gfCNCPoint6[6065] = {X 274.4972, Y 101.6039, Z -8.0000, A 0.000, B 0.000, C 0.000 }
gfCNCPoint6[6066] = {X 273.7387, Y 101.1273, Z -8.0000, A 0.000, B 0.000, C 0.000 }
gfCNCPoint6[6067] = {X 273.1054, Y 100.4940, Z -8.0000, A 0.000, B 0.000, C 0.000 }
gfCNCPoint6[6068] = {X 272.6288, Y 99.7355, Z -8.0000, A 0.000, B 0.000, C 0.000 }
gfCNCPoint6[6069] = {X 272.3330, Y 98.8901, Z -8.0000, A 0.000, B 0.000, C 0.000 }
gfCNCPoint6[6070] = {X 272.2327, Y 98.0000, Z -8.0000, A 0.000, B 0.000, C 0.000 }
gfCNCPoint6[6071] = {X 272.2329, Y 97.0232, Z -8.0000, A 0.000, B 0.000, C 0.000 }
gfCNCPoint6[6072] = {X 272.3321, Y 96.1797, Z -8.0000, A 0.000, B 0.000, C 0.000 }
gfCNCPoint6[6073] = {X 272.6072, Y 95.3761, Z -8.0000, A 0.000, B 0.000, C 0.000 }
gfCNCPoint6[6074] = {X 273.0457, Y 94.6486, Z -8.0000, A 0.000, B 0.000, C 0.000 }
gfCNCPoint6[6075] = {X 273.6280, Y 94.0302, Z -8.0000, A 0.000, B 0.000, C 0.000 }
gfCNCPoint6[6076] = {X 274.3277, Y 93.5487, Z -8.0000, A 0.000, B 0.000, C 0.000 }
gfCNCPoint6[6077] = {X 275.1133, Y 93.2258, Z -8.0000, A 0.000, B 0.000, C 0.000 }
gfCNCPoint6[6078] = {X 275.9494, Y 93.0760, Z -8.0000, A 0.000, B 0.000, C 0.000 }
gfCNCPoint6[6079] = {X 275.9494, Y 85.3767, Z -8.0000, A 0.000, B 0.000, C 0.000 }
gfCNCPoint6[6080] = {X 262.6059, Y 80.1460, Z -8.0000, A 0.000, B 0.000, C 0.000 }
gfCNCPoint6[6081] = {X 237.4769, Y 96.4149, Z -8.0000, A 0.000, B 0.000, C 0.000 }
gfCNCPoint6[6082] = {X 237.4798, Y 97.0659, Z -8.0000, A 0.000, B 0.000, C 0.000 }
gfCNCPoint6[6083] = {X 237.4798, Y 98.0000, Z -8.0000, A 0.000, B 0.000, C 0.000 }
gfCNCPoint6[6084] = {X 237.3795, Y 98.8901, Z -8.0000, A 0.000, B 0.000, C 0.000 }
gfCNCPoint6[6085] = {X 237.0837, Y 99.7355, Z -8.0000, A 0.000, B 0.000, C 0.000 }
gfCNCPoint6[6086] = {X 236.6071, Y 100.4940, Z -8.0000, A 0.000, B 0.000, C 0.000 }
gfCNCPoint6[6087] = {X 235.9737, Y 101.1273, Z -8.0000, A 0.000, B 0.000, C 0.000 }
gfCNCPoint6[6088] = {X 235.2153, Y 101.6039, Z -8.0000, A 0.000, B 0.000, C 0.000 }
gfCNCPoint6[6089] = {X 234.3699, Y 101.8997, Z -8.0000, A 0.000, B 0.000, C 0.000 }
gfCNCPoint6[6090] = {X 233.4798, Y 102.0000, Z -8.0000, A 0.000, B 0.000, C 0.000 }
gfCNCPoint6[6091] = {X 214.1790, Y 102.0000, Z -8.0000, A 0.000, B 0.000, C 0.000 }
gfCNCPoint6[6092] = {X 213.7859, Y 101.9806, Z -8.0000, A 0.000, B 0.000, C 0.000 }
gfCNCPoint6[6093] = {X 213.3966, Y 101.9227, Z -8.0000, A 0.000, B 0.000, C 0.000 }
gfCNCPoint6[6094] = {X 213.0072, Y 101.9806, Z -8.0000, A 0.000, B 0.000, C 0.000 }
gfCNCPoint6[6095] = {X 212.6141, Y 102.0000, Z -8.0000, A 0.000, B 0.000, C 0.000 }
gfCNCPoint6[6096] = {X 194.9870, Y 102.0000, Z -8.0000, A 0.000, B 0.000, C 0.000 }
gfCNCPoint6[6097] = {X 194.0969, Y 101.8997, Z -8.0000, A 0.000, B 0.000, C 0.000 }
gfCNCPoint6[6098] = {X 193.2514, Y 101.6039, Z -8.0000, A 0.000, B 0.000, C 0.000 }
gfCNCPoint6[6099] = {X 192.4930, Y 101.1273, Z -8.0000, A 0.000, B 0.000, C 0.000 }
gfCNCPoint6[6100] = {X 191.8596, Y 100.4940, Z -8.0000, A 0.000, B 0.000, C 0.000 }
gfCNCPoint6[6101] = {X 191.3831, Y 99.7355, Z -8.0000, A 0.000, B 0.000, C 0.000 }
gfCNCPoint6[6102] = {X 191.0872, Y 98.8901, Z -8.0000, A 0.000, B 0.000, C 0.000 }
gfCNCPoint6[6103] = {X 190.9870, Y 98.0000, Z -8.0000, A 0.000, B 0.000, C 0.000 }
gfCNCPoint6[6104] = {X 190.9870, Y 97.0659, Z -8.0000, A 0.000, B 0.000, C 0.000 }
gfCNCPoint6[6105] = {X 191.0804, Y 96.2066, Z -8.0000, A 0.000, B 0.000, C 0.000 }
gfCNCPoint6[6106] = {X 191.3562, Y 95.3874, Z -8.0000, A 0.000, B 0.000, C 0.000 }
gfCNCPoint6[6107] = {X 191.8015, Y 94.6466, Z -8.0000, A 0.000, B 0.000, C 0.000 }
gfCNCPoint6[6108] = {X 191.9051, Y 94.5173, Z -8.0000, A 0.000, B 0.000, C 0.000 }
gfCNCPoint6[6109] = {X 192.0141, Y 94.3923, Z -8.0000, A 0.000, B 0.000, C 0.000 }
gfCNCPoint6[6110] = {X 188.7055, Y 90.7802, Z -8.0000, A 0.000, B 0.000, C 0.000 }
gfCNCPoint6[6111] = {X 149.9476, Y 90.7802, Z -8.0000, A 0.000, B 0.000, C 0.000 }
gfCNCPoint6[6112] = {X 146.7195, Y 94.3565, Z -8.0000, A 0.000, B 0.000, C 0.000 }
gfCNCPoint6[6113] = {X 147.1699, Y 94.9478, Z -8.0000, A 0.000, B 0.000, C 0.000 }
gfCNCPoint6[6114] = {X 147.5035, Y 95.6119, Z -8.0000, A 0.000, B 0.000, C 0.000 }
gfCNCPoint6[6115] = {X 147.7089, Y 96.3261, Z -8.0000, A 0.000, B 0.000, C 0.000 }
gfCNCPoint6[6116] = {X 147.7791, Y 97.0660, Z -8.0000, A 0.000, B 0.000, C 0.000 }
gfCNCPoint6[6117] = {X 147.7791, Y 98.0000, Z -8.0000, A 0.000, B 0.000, C 0.000 }
gfCNCPoint6[6118] = {X 147.6788, Y 98.8901, Z -8.0000, A 0.000, B 0.000, C 0.000 }
gfCNCPoint6[6119] = {X 147.3830, Y 99.7355, Z -8.0000, A 0.000, B 0.000, C 0.000 }
gfCNCPoint6[6120] = {X 146.9064, Y 100.4940, Z -8.0000, A 0.000, B 0.000, C 0.000 }
gfCNCPoint6[6121] = {X 146.2731, Y 101.1273, Z -8.0000, A 0.000, B 0.000, C 0.000 }
gfCNCPoint6[6122] = {X 145.5146, Y 101.6039, Z -8.0000, A 0.000, B 0.000, C 0.000 }
gfCNCPoint6[6123] = {X 144.6692, Y 101.8997, Z -8.0000, A 0.000, B 0.000, C 0.000 }
gfCNCPoint6[6124] = {X 143.7791, Y 102.0000, Z -8.0000, A 0.000, B 0.000, C 0.000 }
gfCNCPoint6[6125] = {X 125.0000, Y 102.0000, Z -8.0000, A 0.000, B 0.000, C 0.000 }
gfCNCPoint6[6126] = {X 124.1099, Y 101.8997, Z -8.0000, A 0.000, B 0.000, C 0.000 }
gfCNCPoint6[6127] = {X 123.2645, Y 101.6039, Z -8.0000, A 0.000, B 0.000, C 0.000 }
gfCNCPoint6[6128] = {X 122.5060, Y 101.1273, Z -8.0000, A 0.000, B 0.000, C 0.000 }
gfCNCPoint6[6129] = {X 121.8727, Y 100.4940, Z -8.0000, A 0.000, B 0.000, C 0.000 }
gfCNCPoint6[6130] = {X 121.3961, Y 99.7355, Z -8.0000, A 0.000, B 0.000, C 0.000 }
gfCNCPoint6[6131] = {X 121.1003, Y 98.8901, Z -8.0000, A 0.000, B 0.000, C 0.000 }
gfCNCPoint6[6132] = {X 121.0000, Y 98.0000, Z -8.0000, A 0.000, B 0.000, C 0.000 }
gfCNCPoint6[6133] = {X 121.0000, Y 97.0659, Z -8.0000, A 0.000, B 0.000, C 0.000 }
gfCNCPoint6[6134] = {X 121.0981, Y 96.1853, Z -8.0000, A 0.000, B 0.000, C 0.000 }
gfCNCPoint6[6135] = {X 121.3877, Y 95.3479, Z -8.0000, A 0.000, B 0.000, C 0.000 }
gfCNCPoint6[6136] = {X 121.8546, Y 94.5948, Z -8.0000, A 0.000, B 0.000, C 0.000 }
gfCNCPoint6[6137] = {X 122.4758, Y 93.9629, Z -8.0000, A 0.000, B 0.000, C 0.000 }
gfCNCPoint6[6138] = {X 123.2209, Y 93.4834, Z -8.0000, A 0.000, B 0.000, C 0.000 }
gfCNCPoint6[6139] = {X 124.0533, Y 93.1796, Z -8.0000, A 0.000, B 0.000, C 0.000 }
gfCNCPoint6[6140] = {X 124.9321, Y 93.0665, Z -8.0000, A 0.000, B 0.000, C 0.000 }
gfCNCPoint6[6141] = {X 124.9746, Y 93.0367, Z -8.0000, A 0.000, B 0.000, C 0.000 }
gfCNCPoint6[6142] = {X 125.4940, Y 92.9596, Z -8.0000, A 0.000, B 0.000, C 0.000 }
gfCNCPoint6[6143] = {X 126.3820, Y 92.8084, Z -8.0000, A 0.000, B 0.000, C 0.000 }
gfCNCPoint6[6144] = {X 127.2570, Y 92.5949, Z -8.0000, A 0.000, B 0.000, C 0.000 }
gfCNCPoint6[6145] = {X 128.4861, Y 91.4437, Z -8.0000, A 0.000, B 0.000, C 0.000 }
gfCNCPoint6[6146] = {X 129.6489, Y 90.2255, Z -8.0000, A 0.000, B 0.000, C 0.000 }
gfCNCPoint6[6147] = {X 140.9159, Y 77.8537, Z -8.0000, A 0.000, B 0.000, C 0.000 }
gfCNCPoint6[6148] = {X 137.8994, Y 75.1065, Z -8.0000, A 0.000, B 0.000, C 0.000 }
gfCNCPoint6[6149] = {X 137.8994, Y 75.1065, Z -5.0000, A 0.000, B 0.000, C 0.000 }
gfCNCPoint6[6150] = {X 137.8994, Y 75.1065, Z 11.0000, A 0.000, B 0.000, C 0.000 }
gfCNCPoint6[6151] = {X 165.2857, Y 38.5771, Z 11.0000, A 0.000, B 0.000, C 0.000 }
gfCNCPoint6[6152] = {X 165.2857, Y 38.5771, Z -5.0000, A 0.000, B 0.000, C 0.000 }
gfCNCPoint6[6153] = {X 165.2857, Y 38.5771, Z -8.0000, A 0.000, B 0.000, C 0.000 }
gfCNCPoint6[6154] = {X 169.3150, Y 37.9356, Z -8.0000, A 0.000, B 0.000, C 0.000 }
gfCNCPoint6[6155] = {X 169.2595, Y 37.5870, Z -8.0000, A 0.000, B 0.000, C 0.000 }
gfCNCPoint6[6156] = {X 169.1010, Y 35.9822, Z -8.0000, A 0.000, B 0.000, C 0.000 }
gfCNCPoint6[6157] = {X 169.1179, Y 34.3697, Z -8.0000, A 0.000, B 0.000, C 0.000 }
gfCNCPoint6[6158] = {X 169.3102, Y 32.7686, Z -8.0000, A 0.000, B 0.000, C 0.000 }
gfCNCPoint6[6159] = {X 169.6755, Y 31.1979, Z -8.0000, A 0.000, B 0.000, C 0.000 }
gfCNCPoint6[6160] = {X 170.2095, Y 29.6763, Z -8.0000, A 0.000, B 0.000, C 0.000 }
gfCNCPoint6[6161] = {X 170.8480, Y 28.3694, Z -8.0000, A 0.000, B 0.000, C 0.000 }
gfCNCPoint6[6162] = {X 171.6556, Y 27.1596, Z -8.0000, A 0.000, B 0.000, C 0.000 }
gfCNCPoint6[6163] = {X 172.6177, Y 26.0688, Z -8.0000, A 0.000, B 0.000, C 0.000 }
gfCNCPoint6[6164] = {X 173.7171, Y 25.1164, Z -8.0000, A 0.000, B 0.000, C 0.000 }
gfCNCPoint6[6165] = {X 174.9340, Y 24.3195, Z -8.0000, A 0.000, B 0.000, C 0.000 }
gfCNCPoint6[6166] = {X 174.1517, Y 23.9319, Z -8.0000, A 0.000, B 0.000, C 0.000 }
gfCNCPoint6[6167] = {X 173.4633, Y 23.3948, Z -8.0000, A 0.000, B 0.000, C 0.000 }
gfCNCPoint6[6168] = {X 172.8970, Y 22.7303, Z -8.0000, A 0.000, B 0.000, C 0.000 }
gfCNCPoint6[6169] = {X 172.4758, Y 21.9655, Z -8.0000, A 0.000, B 0.000, C 0.000 }
gfCNCPoint6[6170] = {X 169.8405, Y 15.5121, Z -8.0000, A 0.000, B 0.000, C 0.000 }
gfCNCPoint6[6171] = {X 169.5912, Y 14.6607, Z -8.0000, A 0.000, B 0.000, C 0.000 }
gfCNCPoint6[6172] = {X 169.5212, Y 13.7764, Z -8.0000, A 0.000, B 0.000, C 0.000 }
gfCNCPoint6[6173] = {X 169.6332, Y 12.8964, Z -8.0000, A 0.000, B 0.000, C 0.000 }
gfCNCPoint6[6174] = {X 169.9226, Y 12.0578, Z -8.0000, A 0.000, B 0.000, C 0.000 }
gfCNCPoint6[6175] = {X 170.3773, Y 11.2960, Z -8.0000, A 0.000, B 0.000, C 0.000 }
gfCNCPoint6[6176] = {X 170.9779, Y 10.6432, Z -8.0000, A 0.000, B 0.000, C 0.000 }
gfCNCPoint6[6177] = {X 171.6992, Y 10.1268, Z -8.0000, A 0.000, B 0.000, C 0.000 }
gfCNCPoint6[6178] = {X 172.3295, Y 9.7674, Z -8.0000, A 0.000, B 0.000, C 0.000 }
gfCNCPoint6[6179] = {X 173.1918, Y 9.4018, Z -8.0000, A 0.000, B 0.000, C 0.000 }
gfCNCPoint6[6180] = {X 174.1126, Y 9.2307, Z -8.0000, A 0.000, B 0.000, C 0.000 }
gfCNCPoint6[6181] = {X 175.0486, Y 9.2620, Z -8.0000, A 0.000, B 0.000, C 0.000 }
gfCNCPoint6[6182] = {X 175.9559, Y 9.4943, Z -8.0000, A 0.000, B 0.000, C 0.000 }
gfCNCPoint6[6183] = {X 177.1286, Y 9.0434, Z -8.0000, A 0.000, B 0.000, C 0.000 }
gfCNCPoint6[6184] = {X 179.2966, Y 8.2457, Z -8.0000, A 0.000, B 0.000, C 0.000 }
gfCNCPoint6[6185] = {X 181.5326, Y 7.6654, Z -8.0000, A 0.000, B 0.000, C 0.000 }
gfCNCPoint6[6186] = {X 183.8149, Y 7.3083, Z -8.0000, A 0.000, B 0.000, C 0.000 }
gfCNCPoint6[6187] = {X 186.1213, Y 7.1778, Z -8.0000, A 0.000, B 0.000, C 0.000 }
gfCNCPoint6[6188] = {X 188.4294, Y 7.2751, Z -8.0000, A 0.000, B 0.000, C 0.000 }
gfCNCPoint6[6189] = {X 190.7166, Y 7.5994, Z -8.0000, A 0.000, B 0.000, C 0.000 }
gfCNCPoint6[6190] = {X 192.3080, Y 7.9856, Z -8.0000, A 0.000, B 0.000, C 0.000 }
gfCNCPoint6[6191] = {X 193.8552, Y 8.5222, Z -8.0000, A 0.000, B 0.000, C 0.000 }
gfCNCPoint6[6192] = {X 195.3440, Y 9.2045, Z -8.0000, A 0.000, B 0.000, C 0.000 }
gfCNCPoint6[6193] = {X 196.7606, Y 10.0260, Z -8.0000, A 0.000, B 0.000, C 0.000 }
gfCNCPoint6[6194] = {X 198.0922, Y 10.9792, Z -8.0000, A 0.000, B 0.000, C 0.000 }
gfCNCPoint6[6195] = {X 199.1520, Y 11.9221, Z -8.0000, A 0.000, B 0.000, C 0.000 }
gfCNCPoint6[6196] = {X 200.1030, Y 12.9747, Z -8.0000, A 0.000, B 0.000, C 0.000 }
gfCNCPoint6[6197] = {X 200.9339, Y 14.1244, Z -8.0000, A 0.000, B 0.000, C 0.000 }
gfCNCPoint6[6198] = {X 201.6348, Y 15.3577, Z -8.0000, A 0.000, B 0.000, C 0.000 }
gfCNCPoint6[6199] = {X 202.1974, Y 16.6600, Z -8.0000, A 0.000, B 0.000, C 0.000 }
gfCNCPoint6[6200] = {X 202.6716, Y 18.3163, Z -8.0000, A 0.000, B 0.000, C 0.000 }
gfCNCPoint6[6201] = {X 202.9530, Y 20.0160, Z -8.0000, A 0.000, B 0.000, C 0.000 }
gfCNCPoint6[6202] = {X 203.0380, Y 21.7368, Z -8.0000, A 0.000, B 0.000, C 0.000 }
gfCNCPoint6[6203] = {X 202.9255, Y 23.4560, Z -8.0000, A 0.000, B 0.000, C 0.000 }
gfCNCPoint6[6204] = {X 202.6168, Y 25.1510, Z -8.0000, A 0.000, B 0.000, C 0.000 }
gfCNCPoint6[6205] = {X 202.1749, Y 26.5972, Z -8.0000, A 0.000, B 0.000, C 0.000 }
gfCNCPoint6[6206] = {X 201.5500, Y 27.9742, Z -8.0000, A 0.000, B 0.000, C 0.000 }
gfCNCPoint6[6207] = {X 200.7528, Y 29.2592, Z -8.0000, A 0.000, B 0.000, C 0.000 }
gfCNCPoint6[6208] = {X 199.7964, Y 30.4306, Z -8.0000, A 0.000, B 0.000, C 0.000 }
gfCNCPoint6[6209] = {X 198.6969, Y 31.4688, Z -8.0000, A 0.000, B 0.000, C 0.000 }
gfCNCPoint6[6210] = {X 199.4979, Y 31.8101, Z -8.0000, A 0.000, B 0.000, C 0.000 }
gfCNCPoint6[6211] = {X 200.2141, Y 32.3050, Z -8.0000, A 0.000, B 0.000, C 0.000 }
gfCNCPoint6[6212] = {X 200.8166, Y 32.9336, Z -8.0000, A 0.000, B 0.000, C 0.000 }
gfCNCPoint6[6213] = {X 201.2808, Y 33.6702, Z -8.0000, A 0.000, B 0.000, C 0.000 }
gfCNCPoint6[6214] = {X 204.3222, Y 39.9530, Z -8.0000, A 0.000, B 0.000, C 0.000 }
gfCNCPoint6[6215] = {X 204.6427, Y 40.8622, Z -8.0000, A 0.000, B 0.000, C 0.000 }
gfCNCPoint6[6216] = {X 204.7537, Y 41.8197, Z -8.0000, A 0.000, B 0.000, C 0.000 }
gfCNCPoint6[6217] = {X 204.6496, Y 42.7781, Z -8.0000, A 0.000, B 0.000, C 0.000 }
gfCNCPoint6[6218] = {X 204.3355, Y 43.6895, Z -8.0000, A 0.000, B 0.000, C 0.000 }
gfCNCPoint6[6219] = {X 203.8272, Y 44.5085, Z -8.0000, A 0.000, B 0.000, C 0.000 }
gfCNCPoint6[6220] = {X 203.1499, Y 45.1945, Z -8.0000, A 0.000, B 0.000, C 0.000 }
gfCNCPoint6[6221] = {X 202.6139, Y 45.6278, Z -8.0000, A 0.000, B 0.000, C 0.000 }
gfCNCPoint6[6222] = {X 201.9096, Y 46.0923, Z -8.0000, A 0.000, B 0.000, C 0.000 }
gfCNCPoint6[6223] = {X 201.1286, Y 46.4113, Z -8.0000, A 0.000, B 0.000, C 0.000 }
gfCNCPoint6[6224] = {X 200.3005, Y 46.5727, Z -8.0000, A 0.000, B 0.000, C 0.000 }
gfCNCPoint6[6225] = {X 199.4569, Y 46.5704, Z -8.0000, A 0.000, B 0.000, C 0.000 }
gfCNCPoint6[6226] = {X 198.6297, Y 46.4045, Z -8.0000, A 0.000, B 0.000, C 0.000 }
gfCNCPoint6[6227] = {X 196.5191, Y 47.5053, Z -8.0000, A 0.000, B 0.000, C 0.000 }
gfCNCPoint6[6228] = {X 194.3239, Y 48.4257, Z -8.0000, A 0.000, B 0.000, C 0.000 }
gfCNCPoint6[6229] = {X 192.0594, Y 49.1592, Z -8.0000, A 0.000, B 0.000, C 0.000 }
gfCNCPoint6[6230] = {X 189.8462, Y 49.6717, Z -8.0000, A 0.000, B 0.000, C 0.000 }
gfCNCPoint6[6231] = {X 187.5926, Y 49.9576, Z -8.0000, A 0.000, B 0.000, C 0.000 }
gfCNCPoint6[6232] = {X 185.3216, Y 50.0138, Z -8.0000, A 0.000, B 0.000, C 0.000 }
gfCNCPoint6[6233] = {X 183.0565, Y 49.8399, Z -8.0000, A 0.000, B 0.000, C 0.000 }
gfCNCPoint6[6234] = {X 180.8207, Y 49.4375, Z -8.0000, A 0.000, B 0.000, C 0.000 }
gfCNCPoint6[6235] = {X 178.9807, Y 48.9033, Z -8.0000, A 0.000, B 0.000, C 0.000 }
gfCNCPoint6[6236] = {X 177.2144, Y 48.1610, Z -8.0000, A 0.000, B 0.000, C 0.000 }
gfCNCPoint6[6237] = {X 175.5452, Y 47.2205, Z -8.0000, A 0.000, B 0.000, C 0.000 }
gfCNCPoint6[6238] = {X 173.9952, Y 46.0942, Z -8.0000, A 0.000, B 0.000, C 0.000 }
gfCNCPoint6[6239] = {X 172.8545, Y 45.0533, Z -8.0000, A 0.000, B 0.000, C 0.000 }
gfCNCPoint6[6240] = {X 171.8449, Y 43.8848, Z -8.0000, A 0.000, B 0.000, C 0.000 }
gfCNCPoint6[6241] = {X 170.9807, Y 42.6050, Z -8.0000, A 0.000, B 0.000, C 0.000 }
gfCNCPoint6[6242] = {X 170.2740, Y 41.2319, Z -8.0000, A 0.000, B 0.000, C 0.000 }
gfCNCPoint6[6243] = {X 169.7348, Y 39.7849, Z -8.0000, A 0.000, B 0.000, C 0.000 }
gfCNCPoint6[6244] = {X 169.3705, Y 38.2842, Z -8.0000, A 0.000, B 0.000, C 0.000 }
gfCNCPoint6[6245] = {X 169.3150, Y 37.9356, Z -8.0000, A 0.000, B 0.000, C 0.000 }
gfCNCPoint6[6246] = {X 165.3647, Y 38.5646, Z -8.0000, A 0.000, B 0.000, C 0.000 }
gfCNCPoint6[6247] = {X 169.3940, Y 37.9231, Z -8.0000, A 0.000, B 0.000, C 0.000 }
gfCNCPoint6[6248] = {X 169.3385, Y 37.5748, Z -8.0000, A 0.000, B 0.000, C 0.000 }
gfCNCPoint6[6249] = {X 169.1809, Y 35.9787, Z -8.0000, A 0.000, B 0.000, C 0.000 }
gfCNCPoint6[6250] = {X 169.1978, Y 34.3748, Z -8.0000, A 0.000, B 0.000, C 0.000 }
gfCNCPoint6[6251] = {X 169.3890, Y 32.7823, Z -8.0000, A 0.000, B 0.000, C 0.000 }
gfCNCPoint6[6252] = {X 169.7524, Y 31.2201, Z -8.0000, A 0.000, B 0.000, C 0.000 }
gfCNCPoint6[6253] = {X 170.2835, Y 29.7067, Z -8.0000, A 0.000, B 0.000, C 0.000 }
gfCNCPoint6[6254] = {X 170.9351, Y 28.3785, Z -8.0000, A 0.000, B 0.000, C 0.000 }
gfCNCPoint6[6255] = {X 171.7625, Y 27.1522, Z -8.0000, A 0.000, B 0.000, C 0.000 }
gfCNCPoint6[6256] = {X 172.7502, Y 26.0509, Z -8.0000, A 0.000, B 0.000, C 0.000 }
gfCNCPoint6[6257] = {X 173.8794, Y 25.0952, Z -8.0000, A 0.000, B 0.000, C 0.000 }
gfCNCPoint6[6258] = {X 175.1290, Y 24.3033, Z -8.0000, A 0.000, B 0.000, C 0.000 }
gfCNCPoint6[6259] = {X 174.3078, Y 23.9331, Z -8.0000, A 0.000, B 0.000, C 0.000 }
gfCNCPoint6[6260] = {X 173.5833, Y 23.3977, Z -8.0000, A 0.000, B 0.000, C 0.000 }
gfCNCPoint6[6261] = {X 172.9883, Y 22.7214, Z -8.0000, A 0.000, B 0.000, C 0.000 }
gfCNCPoint6[6262] = {X 172.5496, Y 21.9347, Z -8.0000, A 0.000, B 0.000, C 0.000 }
gfCNCPoint6[6263] = {X 169.9145, Y 15.4818, Z -8.0000, A 0.000, B 0.000, C 0.000 }
gfCNCPoint6[6264] = {X 169.6699, Y 14.6462, Z -8.0000, A 0.000, B 0.000, C 0.000 }
gfCNCPoint6[6265] = {X 169.6011, Y 13.7783, Z -8.0000, A 0.000, B 0.000, C 0.000 }
gfCNCPoint6[6266] = {X 169.7111, Y 12.9146, Z -8.0000, A 0.000, B 0.000, C 0.000 }
gfCNCPoint6[6267] = {X 169.9952, Y 12.0915, Z -8.0000, A 0.000, B 0.000, C 0.000 }
gfCNCPoint6[6268] = {X 170.4414, Y 11.3439, Z -8.0000, A 0.000, B 0.000, C 0.000 }
gfCNCPoint6[6269] = {X 171.0309, Y 10.7031, Z -8.0000, A 0.000, B 0.000, C 0.000 }
gfCNCPoint6[6270] = {X 171.7389, Y 10.1963, Z -8.0000, A 0.000, B 0.000, C 0.000 }
gfCNCPoint6[6271] = {X 172.3689, Y 9.8371, Z -8.0000, A 0.000, B 0.000, C 0.000 }
gfCNCPoint6[6272] = {X 173.2224, Y 9.4762, Z -8.0000, A 0.000, B 0.000, C 0.000 }
gfCNCPoint6[6273] = {X 174.1339, Y 9.3093, Z -8.0000, A 0.000, B 0.000, C 0.000 }
gfCNCPoint6[6274] = {X 175.0599, Y 9.3445, Z -8.0000, A 0.000, B 0.000, C 0.000 }
gfCNCPoint6[6275] = {X 175.9561, Y 9.5799, Z -8.0000, A 0.000, B 0.000, C 0.000 }
gfCNCPoint6[6276] = {X 177.1586, Y 9.1176, Z -8.0000, A 0.000, B 0.000, C 0.000 }
gfCNCPoint6[6277] = {X 179.3194, Y 8.3224, Z -8.0000, A 0.000, B 0.000, C 0.000 }
gfCNCPoint6[6278] = {X 181.5480, Y 7.7439, Z -8.0000, A 0.000, B 0.000, C 0.000 }
gfCNCPoint6[6279] = {X 183.8227, Y 7.3879, Z -8.0000, A 0.000, B 0.000, C 0.000 }
gfCNCPoint6[6280] = {X 186.1214, Y 7.2578, Z -8.0000, A 0.000, B 0.000, C 0.000 }
gfCNCPoint6[6281] = {X 188.4218, Y 7.3548, Z -8.0000, A 0.000, B 0.000, C 0.000 }
gfCNCPoint6[6282] = {X 190.7015, Y 7.6779, Z -8.0000, A 0.000, B 0.000, C 0.000 }
gfCNCPoint6[6283] = {X 192.2855, Y 8.0623, Z -8.0000, A 0.000, B 0.000, C 0.000 }
gfCNCPoint6[6284] = {X 193.8254, Y 8.5965, Z -8.0000, A 0.000, B 0.000, C 0.000 }
gfCNCPoint6[6285] = {X 195.3072, Y 9.2755, Z -8.0000, A 0.000, B 0.000, C 0.000 }
gfCNCPoint6[6286] = {X 196.7172, Y 10.0932, Z -8.0000, A 0.000, B 0.000, C 0.000 }
gfCNCPoint6[6287] = {X 198.0426, Y 11.0420, Z -8.0000, A 0.000, B 0.000, C 0.000 }
gfCNCPoint6[6288] = {X 199.0958, Y 11.9791, Z -8.0000, A 0.000, B 0.000, C 0.000 }
gfCNCPoint6[6289] = {X 200.0409, Y 13.0251, Z -8.0000, A 0.000, B 0.000, C 0.000 }
gfCNCPoint6[6290] = {X 200.8666, Y 14.1678, Z -8.0000, A 0.000, B 0.000, C 0.000 }
gfCNCPoint6[6291] = {X 201.5632, Y 15.3935, Z -8.0000, A 0.000, B 0.000, C 0.000 }
gfCNCPoint6[6292] = {X 202.1223, Y 16.6876, Z -8.0000, A 0.000, B 0.000, C 0.000 }
gfCNCPoint6[6293] = {X 202.5938, Y 18.3350, Z -8.0000, A 0.000, B 0.000, C 0.000 }
gfCNCPoint6[6294] = {X 202.8736, Y 20.0255, Z -8.0000, A 0.000, B 0.000, C 0.000 }
gfCNCPoint6[6295] = {X 202.9580, Y 21.7368, Z -8.0000, A 0.000, B 0.000, C 0.000 }
gfCNCPoint6[6296] = {X 202.8460, Y 23.4467, Z -8.0000, A 0.000, B 0.000, C 0.000 }
gfCNCPoint6[6297] = {X 202.5390, Y 25.1324, Z -8.0000, A 0.000, B 0.000, C 0.000 }
gfCNCPoint6[6298] = {X 202.0893, Y 26.5970, Z -8.0000, A 0.000, B 0.000, C 0.000 }
gfCNCPoint6[6299] = {X 201.4509, Y 27.9898, Z -8.0000, A 0.000, B 0.000, C 0.000 }
gfCNCPoint6[6300] = {X 200.6347, Y 29.2864, Z -8.0000, A 0.000, B 0.000, C 0.000 }
gfCNCPoint6[6301] = {X 199.6550, Y 30.4643, Z -8.0000, A 0.000, B 0.000, C 0.000 }
gfCNCPoint6[6302] = {X 198.5287, Y 31.5030, Z -8.0000, A 0.000, B 0.000, C 0.000 }
gfCNCPoint6[6303] = {X 199.3597, Y 31.8270, Z -8.0000, A 0.000, B 0.000, C 0.000 }
gfCNCPoint6[6304] = {X 200.1046, Y 32.3177, Z -8.0000, A 0.000, B 0.000, C 0.000 }
gfCNCPoint6[6305] = {X 200.7303, Y 32.9533, Z -8.0000, A 0.000, B 0.000, C 0.000 }
gfCNCPoint6[6306] = {X 201.2091, Y 33.7058, Z -8.0000, A 0.000, B 0.000, C 0.000 }
gfCNCPoint6[6307] = {X 204.2502, Y 39.9879, Z -8.0000, A 0.000, B 0.000, C 0.000 }
gfCNCPoint6[6308] = {X 204.5648, Y 40.8802, Z -8.0000, A 0.000, B 0.000, C 0.000 }
gfCNCPoint6[6309] = {X 204.6737, Y 41.8200, Z -8.0000, A 0.000, B 0.000, C 0.000 }
gfCNCPoint6[6310] = {X 204.5715, Y 42.7606, Z -8.0000, A 0.000, B 0.000, C 0.000 }
gfCNCPoint6[6311] = {X 204.2633, Y 43.6551, Z -8.0000, A 0.000, B 0.000, C 0.000 }
gfCNCPoint6[6312] = {X 203.7643, Y 44.4590, Z -8.0000, A 0.000, B 0.000, C 0.000 }
gfCNCPoint6[6313] = {X 203.0996, Y 45.1323, Z -8.0000, A 0.000, B 0.000, C 0.000 }
gfCNCPoint6[6314] = {X 202.5635, Y 45.5657, Z -8.0000, A 0.000, B 0.000, C 0.000 }
gfCNCPoint6[6315] = {X 201.8662, Y 46.0248, Z -8.0000, A 0.000, B 0.000, C 0.000 }
gfCNCPoint6[6316] = {X 201.0924, Y 46.3386, Z -8.0000, A 0.000, B 0.000, C 0.000 }
gfCNCPoint6[6317] = {X 200.2723, Y 46.4950, Z -8.0000, A 0.000, B 0.000, C 0.000 }
gfCNCPoint6[6318] = {X 199.4374, Y 46.4880, Z -8.0000, A 0.000, B 0.000, C 0.000 }
gfCNCPoint6[6319] = {X 198.6200, Y 46.3178, Z -8.0000, A 0.000, B 0.000, C 0.000 }
gfCNCPoint6[6320] = {X 196.5061, Y 47.4230, Z -8.0000, A 0.000, B 0.000, C 0.000 }
gfCNCPoint6[6321] = {X 194.3068, Y 48.3467, Z -8.0000, A 0.000, B 0.000, C 0.000 }
gfCNCPoint6[6322] = {X 192.0377, Y 49.0822, Z -8.0000, A 0.000, B 0.000, C 0.000 }
gfCNCPoint6[6323] = {X 189.8323, Y 49.5930, Z -8.0000, A 0.000, B 0.000, C 0.000 }
gfCNCPoint6[6324] = {X 187.5867, Y 49.8778, Z -8.0000, A 0.000, B 0.000, C 0.000 }
gfCNCPoint6[6325] = {X 185.3237, Y 49.9339, Z -8.0000, A 0.000, B 0.000, C 0.000 }
gfCNCPoint6[6326] = {X 183.0666, Y 49.7605, Z -8.0000, A 0.000, B 0.000, C 0.000 }
gfCNCPoint6[6327] = {X 180.8387, Y 49.3596, Z -8.0000, A 0.000, B 0.000, C 0.000 }
gfCNCPoint6[6328] = {X 179.0075, Y 48.8279, Z -8.0000, A 0.000, B 0.000, C 0.000 }
gfCNCPoint6[6329] = {X 177.2496, Y 48.0891, Z -8.0000, A 0.000, B 0.000, C 0.000 }
gfCNCPoint6[6330] = {X 175.5883, Y 47.1531, Z -8.0000, A 0.000, B 0.000, C 0.000 }
gfCNCPoint6[6331] = {X 174.0457, Y 46.0322, Z -8.0000, A 0.000, B 0.000, C 0.000 }
gfCNCPoint6[6332] = {X 172.9120, Y 44.9978, Z -8.0000, A 0.000, B 0.000, C 0.000 }
gfCNCPoint6[6333] = {X 171.9087, Y 43.8365, Z -8.0000, A 0.000, B 0.000, C 0.000 }
gfCNCPoint6[6334] = {X 171.0498, Y 42.5647, Z -8.0000, A 0.000, B 0.000, C 0.000 }
gfCNCPoint6[6335] = {X 170.3475, Y 41.2002, Z -8.0000, A 0.000, B 0.000, C 0.000 }
gfCNCPoint6[6336] = {X 169.8115, Y 39.7622, Z -8.0000, A 0.000, B 0.000, C 0.000 }
gfCNCPoint6[6337] = {X 169.4494, Y 38.2708, Z -8.0000, A 0.000, B 0.000, C 0.000 }
gfCNCPoint6[6338] = {X 169.3940, Y 37.9231, Z -8.0000, A 0.000, B 0.000, C 0.000 }
gfCNCPoint6[6339] = {X 165.4437, Y 38.5520, Z -8.0000, A 0.000, B 0.000, C 0.000 }
gfCNCPoint6[6340] = {X 169.4730, Y 37.9105, Z -8.0000, A 0.000, B 0.000, C 0.000 }
gfCNCPoint6[6341] = {X 169.4176, Y 37.5627, Z -8.0000, A 0.000, B 0.000, C 0.000 }
gfCNCPoint6[6342] = {X 169.2608, Y 35.9751, Z -8.0000, A 0.000, B 0.000, C 0.000 }
gfCNCPoint6[6343] = {X 169.2776, Y 34.3799, Z -8.0000, A 0.000, B 0.000, C 0.000 }
gfCNCPoint6[6344] = {X 169.4679, Y 32.7961, Z -8.0000, A 0.000, B 0.000, C 0.000 }
gfCNCPoint6[6345] = {X 169.8292, Y 31.2423, Z -8.0000, A 0.000, B 0.000, C 0.000 }
gfCNCPoint6[6346] = {X 170.3575, Y 29.7370, Z -8.0000, A 0.000, B 0.000, C 0.000 }
gfCNCPoint6[6347] = {X 171.0237, Y 28.3853, Z -8.0000, A 0.000, B 0.000, C 0.000 }
gfCNCPoint6[6348] = {X 171.8734, Y 27.1406, Z -8.0000, A 0.000, B 0.000, C 0.000 }
gfCNCPoint6[6349] = {X 172.8896, Y 26.0278, Z -8.0000, A 0.000, B 0.000, C 0.000 }
gfCNCPoint6[6350] = {X 174.0522, Y 25.0689, Z -8.0000, A 0.000, B 0.000, C 0.000 }
gfCNCPoint6[6351] = {X 175.3381, Y 24.2830, Z -8.0000, A 0.000, B 0.000, C 0.000 }
gfCNCPoint6[6352] = {X 174.4741, Y 23.9349, Z -8.0000, A 0.000, B 0.000, C 0.000 }
gfCNCPoint6[6353] = {X 173.7093, Y 23.4032, Z -8.0000, A 0.000, B 0.000, C 0.000 }
gfCNCPoint6[6354] = {X 173.0819, Y 22.7147, Z -8.0000, A 0.000, B 0.000, C 0.000 }
gfCNCPoint6[6355] = {X 172.6235, Y 21.9039, Z -8.0000, A 0.000, B 0.000, C 0.000 }
gfCNCPoint6[6356] = {X 169.9886, Y 15.4516, Z -8.0000, A 0.000, B 0.000, C 0.000 }
gfCNCPoint6[6357] = {X 169.7252, Y 14.4911, Z -8.0000, A 0.000, B 0.000, C 0.000 }
gfCNCPoint6[6358] = {X 169.6977, Y 13.4955, Z -8.0000, A 0.000, B 0.000, C 0.000 }
gfCNCPoint6[6359] = {X 169.9076, Y 12.5218, Z -8.0000, A 0.000, B 0.000, C 0.000 }
gfCNCPoint6[6360] = {X 170.3429, Y 11.6260, Z -8.0000, A 0.000, B 0.000, C 0.000 }
gfCNCPoint6[6361] = {X 170.9787, Y 10.8594, Z -8.0000, A 0.000, B 0.000, C 0.000 }
gfCNCPoint6[6362] = {X 171.7785, Y 10.2658, Z -8.0000, A 0.000, B 0.000, C 0.000 }
gfCNCPoint6[6363] = {X 172.4082, Y 9.9068, Z -8.0000, A 0.000, B 0.000, C 0.000 }
gfCNCPoint6[6364] = {X 173.2455, Y 9.5528, Z -8.0000, A 0.000, B 0.000, C 0.000 }
gfCNCPoint6[6365] = {X 174.1398, Y 9.3891, Z -8.0000, A 0.000, B 0.000, C 0.000 }
gfCNCPoint6[6366] = {X 175.0482, Y 9.4236, Z -8.0000, A 0.000, B 0.000, C 0.000 }
gfCNCPoint6[6367] = {X 175.9274, Y 9.6546, Z -8.0000, A 0.000, B 0.000, C 0.000 }
gfCNCPoint6[6368] = {X 176.0166, Y 9.6900, Z -8.0000, A 0.000, B 0.000, C 0.000 }
gfCNCPoint6[6369] = {X 177.1899, Y 9.1912, Z -8.0000, A 0.000, B 0.000, C 0.000 }
gfCNCPoint6[6370] = {X 179.3433, Y 8.3987, Z -8.0000, A 0.000, B 0.000, C 0.000 }
gfCNCPoint6[6371] = {X 181.5642, Y 7.8223, Z -8.0000, A 0.000, B 0.000, C 0.000 }
gfCNCPoint6[6372] = {X 183.8312, Y 7.4675, Z -8.0000, A 0.000, B 0.000, C 0.000 }
gfCNCPoint6[6373] = {X 186.1220, Y 7.3378, Z -8.0000, A 0.000, B 0.000, C 0.000 }
gfCNCPoint6[6374] = {X 188.4145, Y 7.4344, Z -8.0000, A 0.000, B 0.000, C 0.000 }
gfCNCPoint6[6375] = {X 190.6863, Y 7.7565, Z -8.0000, A 0.000, B 0.000, C 0.000 }
gfCNCPoint6[6376] = {X 192.2629, Y 8.1391, Z -8.0000, A 0.000, B 0.000, C 0.000 }
gfCNCPoint6[6377] = {X 193.7956, Y 8.6707, Z -8.0000, A 0.000, B 0.000, C 0.000 }
gfCNCPoint6[6378] = {X 195.2704, Y 9.3466, Z -8.0000, A 0.000, B 0.000, C 0.000 }
gfCNCPoint6[6379] = {X 196.6738, Y 10.1604, Z -8.0000, A 0.000, B 0.000, C 0.000 }
gfCNCPoint6[6380] = {X 197.9929, Y 11.1047, Z -8.0000, A 0.000, B 0.000, C 0.000 }
gfCNCPoint6[6381] = {X 199.2848, Y 12.2861, Z -8.0000, A 0.000, B 0.000, C 0.000 }
gfCNCPoint6[6382] = {X 200.4044, Y 13.6319, Z -8.0000, A 0.000, B 0.000, C 0.000 }
gfCNCPoint6[6383] = {X 201.3308, Y 15.1173, Z -8.0000, A 0.000, B 0.000, C 0.000 }
gfCNCPoint6[6384] = {X 202.0470, Y 16.7147, Z -8.0000, A 0.000, B 0.000, C 0.000 }
gfCNCPoint6[6385] = {X 202.5159, Y 18.3531, Z -8.0000, A 0.000, B 0.000, C 0.000 }
gfCNCPoint6[6386] = {X 202.7941, Y 20.0345, Z -8.0000, A 0.000, B 0.000, C 0.000 }
gfCNCPoint6[6387] = {X 202.8780, Y 21.7366, Z -8.0000, A 0.000, B 0.000, C 0.000 }
gfCNCPoint6[6388] = {X 202.7666, Y 23.4371, Z -8.0000, A 0.000, B 0.000, C 0.000 }
gfCNCPoint6[6389] = {X 202.4612, Y 25.1138, Z -8.0000, A 0.000, B 0.000, C 0.000 }
gfCNCPoint6[6390] = {X 202.0032, Y 26.5985, Z -8.0000, A 0.000, B 0.000, C 0.000 }
gfCNCPoint6[6391] = {X 201.3498, Y 28.0081, Z -8.0000, A 0.000, B 0.000, C 0.000 }
gfCNCPoint6[6392] = {X 200.5129, Y 29.3172, Z -8.0000, A 0.000, B 0.000, C 0.000 }
gfCNCPoint6[6393] = {X 199.5077, Y 30.5020, Z -8.0000, A 0.000, B 0.000, C 0.000 }
gfCNCPoint6[6394] = {X 198.3525, Y 31.5410, Z -8.0000, A 0.000, B 0.000, C 0.000 }
gfCNCPoint6[6395] = {X 199.2156, Y 31.8445, Z -8.0000, A 0.000, B 0.000, C 0.000 }
gfCNCPoint6[6396] = {X 199.9914, Y 32.3292, Z -8.0000, A 0.000, B 0.000, C 0.000 }
gfCNCPoint6[6397] = {X 200.6426, Y 32.9719, Z -8.0000, A 0.000, B 0.000, C 0.000 }
gfCNCPoint6[6398] = {X 201.1375, Y 33.7414, Z -8.0000, A 0.000, B 0.000, C 0.000 }
gfCNCPoint6[6399] = {X 204.1781, Y 40.0227, Z -8.0000, A 0.000, B 0.000, C 0.000 }
gfCNCPoint6[6400] = {X 204.4868, Y 40.8982, Z -8.0000, A 0.000, B 0.000, C 0.000 }
gfCNCPoint6[6401] = {X 204.5937, Y 41.8203, Z -8.0000, A 0.000, B 0.000, C 0.000 }
gfCNCPoint6[6402] = {X 204.4934, Y 42.7431, Z -8.0000, A 0.000, B 0.000, C 0.000 }
gfCNCPoint6[6403] = {X 204.1910, Y 43.6208, Z -8.0000, A 0.000, B 0.000, C 0.000 }
gfCNCPoint6[6404] = {X 203.7015, Y 44.4095, Z -8.0000, A 0.000, B 0.000, C 0.000 }
gfCNCPoint6[6405] = {X 203.0493, Y 45.0700, Z -8.0000, A 0.000, B 0.000, C 0.000 }
gfCNCPoint6[6406] = {X 202.5132, Y 45.5035, Z -8.0000, A 0.000, B 0.000, C 0.000 }
gfCNCPoint6[6407] = {X 201.8227, Y 45.9572, Z -8.0000, A 0.000, B 0.000, C 0.000 }
gfCNCPoint6[6408] = {X 201.0564, Y 46.2658, Z -8.0000, A 0.000, B 0.000, C 0.000 }
gfCNCPoint6[6409] = {X 200.2442, Y 46.4172, Z -8.0000, A 0.000, B 0.000, C 0.000 }
gfCNCPoint6[6410] = {X 199.4181, Y 46.4054, Z -8.0000, A 0.000, B 0.000, C 0.000 }
gfCNCPoint6[6411] = {X 198.6105, Y 46.2308, Z -8.0000, A 0.000, B 0.000, C 0.000 }
gfCNCPoint6[6412] = {X 196.4933, Y 47.3406, Z -8.0000, A 0.000, B 0.000, C 0.000 }
gfCNCPoint6[6413] = {X 194.2898, Y 48.2676, Z -8.0000, A 0.000, B 0.000, C 0.000 }
gfCNCPoint6[6414] = {X 192.0160, Y 49.0052, Z -8.0000, A 0.000, B 0.000, C 0.000 }
gfCNCPoint6[6415] = {X 189.8185, Y 49.5142, Z -8.0000, A 0.000, B 0.000, C 0.000 }
gfCNCPoint6[6416] = {X 187.5807, Y 49.7980, Z -8.0000, A 0.000, B 0.000, C 0.000 }
gfCNCPoint6[6417] = {X 185.3258, Y 49.8539, Z -8.0000, A 0.000, B 0.000, C 0.000 }
gfCNCPoint6[6418] = {X 183.0767, Y 49.6812, Z -8.0000, A 0.000, B 0.000, C 0.000 }
gfCNCPoint6[6419] = {X 180.8568, Y 49.2816, Z -8.0000, A 0.000, B 0.000, C 0.000 }
gfCNCPoint6[6420] = {X 179.0343, Y 48.7525, Z -8.0000, A 0.000, B 0.000, C 0.000 }
gfCNCPoint6[6421] = {X 177.2848, Y 48.0173, Z -8.0000, A 0.000, B 0.000, C 0.000 }
gfCNCPoint6[6422] = {X 175.6314, Y 47.0857, Z -8.0000, A 0.000, B 0.000, C 0.000 }
gfCNCPoint6[6423] = {X 174.0962, Y 45.9701, Z -8.0000, A 0.000, B 0.000, C 0.000 }
gfCNCPoint6[6424] = {X 172.9696, Y 44.9422, Z -8.0000, A 0.000, B 0.000, C 0.000 }
gfCNCPoint6[6425] = {X 171.9725, Y 43.7882, Z -8.0000, A 0.000, B 0.000, C 0.000 }
gfCNCPoint6[6426] = {X 171.1189, Y 42.5244, Z -8.0000, A 0.000, B 0.000, C 0.000 }
gfCNCPoint6[6427] = {X 170.4209, Y 41.1684, Z -8.0000, A 0.000, B 0.000, C 0.000 }
gfCNCPoint6[6428] = {X 169.8882, Y 39.7394, Z -8.0000, A 0.000, B 0.000, C 0.000 }
gfCNCPoint6[6429] = {X 169.5282, Y 38.2574, Z -8.0000, A 0.000, B 0.000, C 0.000 }
gfCNCPoint6[6430] = {X 169.4730, Y 37.9105, Z -8.0000, A 0.000, B 0.000, C 0.000 }
gfCNCPoint6[6431] = {X 165.5227, Y 38.5394, Z -8.0000, A 0.000, B 0.000, C 0.000 }
gfCNCPoint6[6432] = {X 169.5520, Y 37.8979, Z -8.0000, A 0.000, B 0.000, C 0.000 }
gfCNCPoint6[6433] = {X 169.4967, Y 37.5505, Z -8.0000, A 0.000, B 0.000, C 0.000 }
gfCNCPoint6[6434] = {X 169.3407, Y 35.9716, Z -8.0000, A 0.000, B 0.000, C 0.000 }
gfCNCPoint6[6435] = {X 169.3575, Y 34.3851, Z -8.0000, A 0.000, B 0.000, C 0.000 }
gfCNCPoint6[6436] = {X 169.5467, Y 32.8098, Z -8.0000, A 0.000, B 0.000, C 0.000 }
gfCNCPoint6[6437] = {X 169.9061, Y 31.2645, Z -8.0000, A 0.000, B 0.000, C 0.000 }
gfCNCPoint6[6438] = {X 170.4315, Y 29.7674, Z -8.0000, A 0.000, B 0.000, C 0.000 }
gfCNCPoint6[6439] = {X 171.1144, Y 28.3888, Z -8.0000, A 0.000, B 0.000, C 0.000 }
gfCNCPoint6[6440] = {X 171.9894, Y 27.1235, Z -8.0000, A 0.000, B 0.000, C 0.000 }
gfCNCPoint6[6441] = {X 173.0383, Y 25.9979, Z -8.0000, A 0.000, B 0.000, C 0.000 }
gfCNCPoint6[6442] = {X 174.2389, Y 25.0359, Z -8.0000, A 0.000, B 0.000, C 0.000 }
gfCNCPoint6[6443] = {X 175.5659, Y 24.2575, Z -8.0000, A 0.000, B 0.000, C 0.000 }
gfCNCPoint6[6444] = {X 174.6541, Y 23.9376, Z -8.0000, A 0.000, B 0.000, C 0.000 }
gfCNCPoint6[6445] = {X 173.8432, Y 23.4123, Z -8.0000, A 0.000, B 0.000, C 0.000 }
gfCNCPoint6[6446] = {X 173.1785, Y 22.7110, Z -8.0000, A 0.000, B 0.000, C 0.000 }
gfCNCPoint6[6447] = {X 172.6973, Y 21.8731, Z -8.0000, A 0.000, B 0.000, C 0.000 }
gfCNCPoint6[6448] = {X 170.0626, Y 15.4213, Z -8.0000, A 0.000, B 0.000, C 0.000 }
gfCNCPoint6[6449] = {X 169.8043, Y 14.4793, Z -8.0000, A 0.000, B 0.000, C 0.000 }
gfCNCPoint6[6450] = {X 169.7773, Y 13.5028, Z -8.0000, A 0.000, B 0.000, C 0.000 }
gfCNCPoint6[6451] = {X 169.9832, Y 12.5479, Z -8.0000, A 0.000, B 0.000, C 0.000 }
gfCNCPoint6[6452] = {X 170.4102, Y 11.6694, Z -8.0000, A 0.000, B 0.000, C 0.000 }
gfCNCPoint6[6453] = {X 171.0337, Y 10.9174, Z -8.0000, A 0.000, B 0.000, C 0.000 }
gfCNCPoint6[6454] = {X 171.8181, Y 10.3353, Z -8.0000, A 0.000, B 0.000, C 0.000 }
gfCNCPoint6[6455] = {X 172.4475, Y 9.9764, Z -8.0000, A 0.000, B 0.000, C 0.000 }
gfCNCPoint6[6456] = {X 173.2687, Y 9.6293, Z -8.0000, A 0.000, B 0.000, C 0.000 }
gfCNCPoint6[6457] = {X 174.1456, Y 9.4689, Z -8.0000, A 0.000, B 0.000, C 0.000 }
gfCNCPoint6[6458] = {X 175.0365, Y 9.5027, Z -8.0000, A 0.000, B 0.000, C 0.000 }
gfCNCPoint6[6459] = {X 175.8988, Y 9.7293, Z -8.0000, A 0.000, B 0.000, C 0.000 }
gfCNCPoint6[6460] = {X 175.9643, Y 9.7551, Z -8.0000, A 0.000, B 0.000, C 0.000 }
gfCNCPoint6[6461] = {X 176.0294, Y 9.7820, Z -8.0000, A 0.000, B 0.000, C 0.000 }
gfCNCPoint6[6462] = {X 176.0570, Y 9.7597, Z -8.0000, A 0.000, B 0.000, C 0.000 }
gfCNCPoint6[6463] = {X 177.2212, Y 9.2648, Z -8.0000, A 0.000, B 0.000, C 0.000 }
gfCNCPoint6[6464] = {X 179.3671, Y 8.4751, Z -8.0000, A 0.000, B 0.000, C 0.000 }
gfCNCPoint6[6465] = {X 181.5805, Y 7.9006, Z -8.0000, A 0.000, B 0.000, C 0.000 }
gfCNCPoint6[6466] = {X 183.8396, Y 7.5470, Z -8.0000, A 0.000, B 0.000, C 0.000 }
gfCNCPoint6[6467] = {X 186.1226, Y 7.4178, Z -8.0000, A 0.000, B 0.000, C 0.000 }
gfCNCPoint6[6468] = {X 188.4072, Y 7.5141, Z -8.0000, A 0.000, B 0.000, C 0.000 }
gfCNCPoint6[6469] = {X 190.6712, Y 7.8350, Z -8.0000, A 0.000, B 0.000, C 0.000 }
gfCNCPoint6[6470] = {X 192.2403, Y 8.2158, Z -8.0000, A 0.000, B 0.000, C 0.000 }
gfCNCPoint6[6471] = {X 193.7658, Y 8.7450, Z -8.0000, A 0.000, B 0.000, C 0.000 }
gfCNCPoint6[6472] = {X 195.2336, Y 9.4176, Z -8.0000, A 0.000, B 0.000, C 0.000 }
gfCNCPoint6[6473] = {X 196.6304, Y 10.2276, Z -8.0000, A 0.000, B 0.000, C 0.000 }
gfCNCPoint6[6474] = {X 197.9433, Y 11.1675, Z -8.0000, A 0.000, B 0.000, C 0.000 }
gfCNCPoint6[6475] = {X 199.2270, Y 12.3413, Z -8.0000, A 0.000, B 0.000, C 0.000 }
gfCNCPoint6[6476] = {X 200.3394, Y 13.6786, Z -8.0000, A 0.000, B 0.000, C 0.000 }
gfCNCPoint6[6477] = {X 201.2600, Y 15.1545, Z -8.0000, A 0.000, B 0.000, C 0.000 }
gfCNCPoint6[6478] = {X 201.9717, Y 16.7417, Z -8.0000, A 0.000, B 0.000, C 0.000 }
gfCNCPoint6[6479] = {X 202.4380, Y 18.3713, Z -8.0000, A 0.000, B 0.000, C 0.000 }
gfCNCPoint6[6480] = {X 202.7146, Y 20.0435, Z -8.0000, A 0.000, B 0.000, C 0.000 }
gfCNCPoint6[6481] = {X 202.7980, Y 21.7363, Z -8.0000, A 0.000, B 0.000, C 0.000 }
gfCNCPoint6[6482] = {X 202.6871, Y 23.4277, Z -8.0000, A 0.000, B 0.000, C 0.000 }
gfCNCPoint6[6483] = {X 202.3834, Y 25.0952, Z -8.0000, A 0.000, B 0.000, C 0.000 }
gfCNCPoint6[6484] = {X 201.9161, Y 26.6018, Z -8.0000, A 0.000, B 0.000, C 0.000 }
gfCNCPoint6[6485] = {X 201.2463, Y 28.0301, Z -8.0000, A 0.000, B 0.000, C 0.000 }
gfCNCPoint6[6486] = {X 200.3866, Y 29.3528, Z -8.0000, A 0.000, B 0.000, C 0.000 }
gfCNCPoint6[6487] = {X 199.3535, Y 30.5448, Z -8.0000, A 0.000, B 0.000, C 0.000 }
gfCNCPoint6[6488] = {X 198.1663, Y 31.5836, Z -8.0000, A 0.000, B 0.000, C 0.000 }
gfCNCPoint6[6489] = {X 199.0638, Y 31.8625, Z -8.0000, A 0.000, B 0.000, C 0.000 }
gfCNCPoint6[6490] = {X 199.8737, Y 32.3394, Z -8.0000, A 0.000, B 0.000, C 0.000 }
gfCNCPoint6[6491] = {X 200.5530, Y 32.9889, Z -8.0000, A 0.000, B 0.000, C 0.000 }
gfCNCPoint6[6492] = {X 201.0657, Y 33.7766, Z -8.0000, A 0.000, B 0.000, C 0.000 }
gfCNCPoint6[6493] = {X 204.1061, Y 40.0576, Z -8.0000, A 0.000, B 0.000, C 0.000 }
gfCNCPoint6[6494] = {X 204.4089, Y 40.9162, Z -8.0000, A 0.000, B 0.000, C 0.000 }
gfCNCPoint6[6495] = {X 204.5137, Y 41.8206, Z -8.0000, A 0.000, B 0.000, C 0.000 }
gfCNCPoint6[6496] = {X 204.4154, Y 42.7257, Z -8.0000, A 0.000, B 0.000, C 0.000 }
gfCNCPoint6[6497] = {X 204.1188, Y 43.5864, Z -8.0000, A 0.000, B 0.000, C 0.000 }
gfCNCPoint6[6498] = {X 203.6387, Y 44.3600, Z -8.0000, A 0.000, B 0.000, C 0.000 }
gfCNCPoint6[6499] = {X 202.9990, Y 45.0078, Z -8.0000, A 0.000, B 0.000, C 0.000 }
gfCNCPoint6[6500] = {X 202.4629, Y 45.4413, Z -8.0000, A 0.000, B 0.000, C 0.000 }
gfCNCPoint6[6501] = {X 201.7794, Y 45.8896, Z -8.0000, A 0.000, B 0.000, C 0.000 }
gfCNCPoint6[6502] = {X 201.0203, Y 46.1929, Z -8.0000, A 0.000, B 0.000, C 0.000 }
gfCNCPoint6[6503] = {X 200.2161, Y 46.3392, Z -8.0000, A 0.000, B 0.000, C 0.000 }
gfCNCPoint6[6504] = {X 199.3989, Y 46.3226, Z -8.0000, A 0.000, B 0.000, C 0.000 }
gfCNCPoint6[6505] = {X 198.6014, Y 46.1437, Z -8.0000, A 0.000, B 0.000, C 0.000 }
gfCNCPoint6[6506] = {X 196.4806, Y 47.2581, Z -8.0000, A 0.000, B 0.000, C 0.000 }
gfCNCPoint6[6507] = {X 194.2729, Y 48.1886, Z -8.0000, A 0.000, B 0.000, C 0.000 }
gfCNCPoint6[6508] = {X 191.9942, Y 48.9282, Z -8.0000, A 0.000, B 0.000, C 0.000 }
gfCNCPoint6[6509] = {X 189.8046, Y 49.4354, Z -8.0000, A 0.000, B 0.000, C 0.000 }
gfCNCPoint6[6510] = {X 187.5748, Y 49.7183, Z -8.0000, A 0.000, B 0.000, C 0.000 }
gfCNCPoint6[6511] = {X 185.3279, Y 49.7739, Z -8.0000, A 0.000, B 0.000, C 0.000 }
gfCNCPoint6[6512] = {X 183.0869, Y 49.6018, Z -8.0000, A 0.000, B 0.000, C 0.000 }
gfCNCPoint6[6513] = {X 180.8748, Y 49.2037, Z -8.0000, A 0.000, B 0.000, C 0.000 }
gfCNCPoint6[6514] = {X 179.0611, Y 48.6771, Z -8.0000, A 0.000, B 0.000, C 0.000 }
gfCNCPoint6[6515] = {X 177.3200, Y 47.9454, Z -8.0000, A 0.000, B 0.000, C 0.000 }
gfCNCPoint6[6516] = {X 175.6746, Y 47.0183, Z -8.0000, A 0.000, B 0.000, C 0.000 }
gfCNCPoint6[6517] = {X 174.1467, Y 45.9081, Z -8.0000, A 0.000, B 0.000, C 0.000 }
gfCNCPoint6[6518] = {X 173.0272, Y 44.8867, Z -8.0000, A 0.000, B 0.000, C 0.000 }
gfCNCPoint6[6519] = {X 172.0363, Y 43.7400, Z -8.0000, A 0.000, B 0.000, C 0.000 }
gfCNCPoint6[6520] = {X 171.1881, Y 42.4841, Z -8.0000, A 0.000, B 0.000, C 0.000 }
gfCNCPoint6[6521] = {X 170.4943, Y 41.1367, Z -8.0000, A 0.000, B 0.000, C 0.000 }
gfCNCPoint6[6522] = {X 169.9649, Y 39.7167, Z -8.0000, A 0.000, B 0.000, C 0.000 }
gfCNCPoint6[6523] = {X 169.6071, Y 38.2440, Z -8.0000, A 0.000, B 0.000, C 0.000 }
gfCNCPoint6[6524] = {X 169.5520, Y 37.8979, Z -8.0000, A 0.000, B 0.000, C 0.000 }
gfCNCPoint6[6525] = {X 165.6018, Y 38.5268, Z -8.0000, A 0.000, B 0.000, C 0.000 }
gfCNCPoint6[6526] = {X 165.6018, Y 38.5269, Z -8.0000, A 0.000, B 0.000, C 0.000 }
gfCNCPoint6[6527] = {X 169.6310, Y 37.8853, Z -8.0000, A 0.000, B 0.000, C 0.000 }
gfCNCPoint6[6528] = {X 169.5757, Y 37.5383, Z -8.0000, A 0.000, B 0.000, C 0.000 }
gfCNCPoint6[6529] = {X 169.4206, Y 35.9680, Z -8.0000, A 0.000, B 0.000, C 0.000 }
gfCNCPoint6[6530] = {X 169.4373, Y 34.3902, Z -8.0000, A 0.000, B 0.000, C 0.000 }
gfCNCPoint6[6531] = {X 169.6255, Y 32.8235, Z -8.0000, A 0.000, B 0.000, C 0.000 }
gfCNCPoint6[6532] = {X 169.9830, Y 31.2867, Z -8.0000, A 0.000, B 0.000, C 0.000 }
gfCNCPoint6[6533] = {X 170.5055, Y 29.7978, Z -8.0000, A 0.000, B 0.000, C 0.000 }
gfCNCPoint6[6534] = {X 171.2080, Y 28.3878, Z -8.0000, A 0.000, B 0.000, C 0.000 }
gfCNCPoint6[6535] = {X 172.1129, Y 27.0984, Z -8.0000, A 0.000, B 0.000, C 0.000 }
gfCNCPoint6[6536] = {X 173.2000, Y 25.9584, Z -8.0000, A 0.000, B 0.000, C 0.000 }
gfCNCPoint6[6537] = {X 174.4450, Y 24.9932, Z -8.0000, A 0.000, B 0.000, C 0.000 }
gfCNCPoint6[6538] = {X 175.8200, Y 24.2246, Z -8.0000, A 0.000, B 0.000, C 0.000 }
gfCNCPoint6[6539] = {X 175.0293, Y 24.0135, Z -8.0000, A 0.000, B 0.000, C 0.000 }
gfCNCPoint6[6540] = {X 174.2982, Y 23.6459, Z -8.0000, A 0.000, B 0.000, C 0.000 }
gfCNCPoint6[6541] = {X 173.6572, Y 23.1372, Z -8.0000, A 0.000, B 0.000, C 0.000 }
gfCNCPoint6[6542] = {X 173.1331, Y 22.5087, Z -8.0000, A 0.000, B 0.000, C 0.000 }
gfCNCPoint6[6543] = {X 172.7479, Y 21.7867, Z -8.0000, A 0.000, B 0.000, C 0.000 }
gfCNCPoint6[6544] = {X 170.1367, Y 15.3911, Z -8.0000, A 0.000, B 0.000, C 0.000 }
gfCNCPoint6[6545] = {X 169.8835, Y 14.4675, Z -8.0000, A 0.000, B 0.000, C 0.000 }
gfCNCPoint6[6546] = {X 169.8570, Y 13.5102, Z -8.0000, A 0.000, B 0.000, C 0.000 }
gfCNCPoint6[6547] = {X 170.0588, Y 12.5740, Z -8.0000, A 0.000, B 0.000, C 0.000 }
gfCNCPoint6[6548] = {X 170.4774, Y 11.7127, Z -8.0000, A 0.000, B 0.000, C 0.000 }
gfCNCPoint6[6549] = {X 171.0888, Y 10.9755, Z -8.0000, A 0.000, B 0.000, C 0.000 }
gfCNCPoint6[6550] = {X 171.8578, Y 10.4048, Z -8.0000, A 0.000, B 0.000, C 0.000 }
gfCNCPoint6[6551] = {X 172.4867, Y 10.0462, Z -8.0000, A 0.000, B 0.000, C 0.000 }
gfCNCPoint6[6552] = {X 173.2917, Y 9.7059, Z -8.0000, A 0.000, B 0.000, C 0.000 }
gfCNCPoint6[6553] = {X 174.1515, Y 9.5487, Z -8.0000, A 0.000, B 0.000, C 0.000 }
gfCNCPoint6[6554] = {X 175.0248, Y 9.5819, Z -8.0000, A 0.000, B 0.000, C 0.000 }
gfCNCPoint6[6555] = {X 175.8701, Y 9.8040, Z -8.0000, A 0.000, B 0.000, C 0.000 }
gfCNCPoint6[6556] = {X 175.9565, Y 9.8383, Z -8.0000, A 0.000, B 0.000, C 0.000 }
gfCNCPoint6[6557] = {X 176.0421, Y 9.8746, Z -8.0000, A 0.000, B 0.000, C 0.000 }
gfCNCPoint6[6558] = {X 176.0986, Y 9.8290, Z -8.0000, A 0.000, B 0.000, C 0.000 }
gfCNCPoint6[6559] = {X 177.2525, Y 9.3384, Z -8.0000, A 0.000, B 0.000, C 0.000 }
gfCNCPoint6[6560] = {X 179.3910, Y 8.5514, Z -8.0000, A 0.000, B 0.000, C 0.000 }
gfCNCPoint6[6561] = {X 181.5967, Y 7.9789, Z -8.0000, A 0.000, B 0.000, C 0.000 }
gfCNCPoint6[6562] = {X 183.8481, Y 7.6266, Z -8.0000, A 0.000, B 0.000, C 0.000 }
gfCNCPoint6[6563] = {X 186.1232, Y 7.4978, Z -8.0000, A 0.000, B 0.000, C 0.000 }
gfCNCPoint6[6564] = {X 188.3999, Y 7.5937, Z -8.0000, A 0.000, B 0.000, C 0.000 }
gfCNCPoint6[6565] = {X 190.6561, Y 7.9136, Z -8.0000, A 0.000, B 0.000, C 0.000 }
gfCNCPoint6[6566] = {X 192.2178, Y 8.2926, Z -8.0000, A 0.000, B 0.000, C 0.000 }
gfCNCPoint6[6567] = {X 193.7360, Y 8.8192, Z -8.0000, A 0.000, B 0.000, C 0.000 }
gfCNCPoint6[6568] = {X 195.1969, Y 9.4886, Z -8.0000, A 0.000, B 0.000, C 0.000 }
gfCNCPoint6[6569] = {X 196.5870, Y 10.2948, Z -8.0000, A 0.000, B 0.000, C 0.000 }
gfCNCPoint6[6570] = {X 197.8937, Y 11.2302, Z -8.0000, A 0.000, B 0.000, C 0.000 }
gfCNCPoint6[6571] = {X 199.1691, Y 12.3966, Z -8.0000, A 0.000, B 0.000, C 0.000 }
gfCNCPoint6[6572] = {X 200.2745, Y 13.7253, Z -8.0000, A 0.000, B 0.000, C 0.000 }
gfCNCPoint6[6573] = {X 201.1892, Y 15.1917, Z -8.0000, A 0.000, B 0.000, C 0.000 }
gfCNCPoint6[6574] = {X 201.8964, Y 16.7687, Z -8.0000, A 0.000, B 0.000, C 0.000 }
gfCNCPoint6[6575] = {X 202.3600, Y 18.3894, Z -8.0000, A 0.000, B 0.000, C 0.000 }
gfCNCPoint6[6576] = {X 202.6351, Y 20.0525, Z -8.0000, A 0.000, B 0.000, C 0.000 }
gfCNCPoint6[6577] = {X 202.7180, Y 21.7361, Z -8.0000, A 0.000, B 0.000, C 0.000 }
gfCNCPoint6[6578] = {X 202.6077, Y 23.4182, Z -8.0000, A 0.000, B 0.000, C 0.000 }
gfCNCPoint6[6579] = {X 202.3056, Y 25.0766, Z -8.0000, A 0.000, B 0.000, C 0.000 }
gfCNCPoint6[6580] = {X 201.8280, Y 26.6077, Z -8.0000, A 0.000, B 0.000, C 0.000 }
gfCNCPoint6[6581] = {X 201.1398, Y 28.0565, Z -8.0000, A 0.000, B 0.000, C 0.000 }
gfCNCPoint6[6582] = {X 200.2547, Y 29.3941, Z -8.0000, A 0.000, B 0.000, C 0.000 }
gfCNCPoint6[6583] = {X 199.1903, Y 30.5939, Z -8.0000, A 0.000, B 0.000, C 0.000 }
gfCNCPoint6[6584] = {X 197.9678, Y 31.6321, Z -8.0000, A 0.000, B 0.000, C 0.000 }
gfCNCPoint6[6585] = {X 198.7291, Y 31.8163, Z -8.0000, A 0.000, B 0.000, C 0.000 }
gfCNCPoint6[6586] = {X 199.4400, Y 32.1453, Z -8.0000, A 0.000, B 0.000, C 0.000 }
gfCNCPoint6[6587] = {X 200.0732, Y 32.6066, Z -8.0000, A 0.000, B 0.000, C 0.000 }
gfCNCPoint6[6588] = {X 200.6042, Y 33.1824, Z -8.0000, A 0.000, B 0.000, C 0.000 }
gfCNCPoint6[6589] = {X 201.0129, Y 33.8507, Z -8.0000, A 0.000, B 0.000, C 0.000 }
gfCNCPoint6[6590] = {X 204.0341, Y 40.0925, Z -8.0000, A 0.000, B 0.000, C 0.000 }
gfCNCPoint6[6591] = {X 204.3309, Y 40.9342, Z -8.0000, A 0.000, B 0.000, C 0.000 }
gfCNCPoint6[6592] = {X 204.4337, Y 41.8209, Z -8.0000, A 0.000, B 0.000, C 0.000 }
gfCNCPoint6[6593] = {X 204.3373, Y 42.7082, Z -8.0000, A 0.000, B 0.000, C 0.000 }
gfCNCPoint6[6594] = {X 204.0465, Y 43.5521, Z -8.0000, A 0.000, B 0.000, C 0.000 }
gfCNCPoint6[6595] = {X 203.5758, Y 44.3105, Z -8.0000, A 0.000, B 0.000, C 0.000 }
gfCNCPoint6[6596] = {X 202.9487, Y 44.9456, Z -8.0000, A 0.000, B 0.000, C 0.000 }
gfCNCPoint6[6597] = {X 202.4125, Y 45.3791, Z -8.0000, A 0.000, B 0.000, C 0.000 }
gfCNCPoint6[6598] = {X 201.7360, Y 45.8220, Z -8.0000, A 0.000, B 0.000, C 0.000 }
gfCNCPoint6[6599] = {X 200.9844, Y 46.1200, Z -8.0000, A 0.000, B 0.000, C 0.000 }
gfCNCPoint6[6600] = {X 200.1883, Y 46.2611, Z -8.0000, A 0.000, B 0.000, C 0.000 }
gfCNCPoint6[6601] = {X 199.3800, Y 46.2396, Z -8.0000, A 0.000, B 0.000, C 0.000 }
gfCNCPoint6[6602] = {X 198.5925, Y 46.0562, Z -8.0000, A 0.000, B 0.000, C 0.000 }
gfCNCPoint6[6603] = {X 196.4682, Y 47.1755, Z -8.0000, A 0.000, B 0.000, C 0.000 }
gfCNCPoint6[6604] = {X 194.2562, Y 48.1094, Z -8.0000, A 0.000, B 0.000, C 0.000 }
gfCNCPoint6[6605] = {X 191.9725, Y 48.8512, Z -8.0000, A 0.000, B 0.000, C 0.000 }
gfCNCPoint6[6606] = {X 189.7907, Y 49.3566, Z -8.0000, A 0.000, B 0.000, C 0.000 }
gfCNCPoint6[6607] = {X 187.5689, Y 49.6385, Z -8.0000, A 0.000, B 0.000, C 0.000 }
gfCNCPoint6[6608] = {X 185.3300, Y 49.6939, Z -8.0000, A 0.000, B 0.000, C 0.000 }
gfCNCPoint6[6609] = {X 183.0969, Y 49.5224, Z -8.0000, A 0.000, B 0.000, C 0.000 }
gfCNCPoint6[6610] = {X 180.8928, Y 49.1257, Z -8.0000, A 0.000, B 0.000, C 0.000 }
gfCNCPoint6[6611] = {X 179.0878, Y 48.6017, Z -8.0000, A 0.000, B 0.000, C 0.000 }
gfCNCPoint6[6612] = {X 177.3551, Y 47.8736, Z -8.0000, A 0.000, B 0.000, C 0.000 }
gfCNCPoint6[6613] = {X 175.7177, Y 46.9510, Z -8.0000, A 0.000, B 0.000, C 0.000 }
gfCNCPoint6[6614] = {X 174.1973, Y 45.8461, Z -8.0000, A 0.000, B 0.000, C 0.000 }
gfCNCPoint6[6615] = {X 173.0848, Y 44.8311, Z -8.0000, A 0.000, B 0.000, C 0.000 }
gfCNCPoint6[6616] = {X 172.1001, Y 43.6917, Z -8.0000, A 0.000, B 0.000, C 0.000 }
gfCNCPoint6[6617] = {X 171.2572, Y 42.4438, Z -8.0000, A 0.000, B 0.000, C 0.000 }
gfCNCPoint6[6618] = {X 170.5678, Y 41.1049, Z -8.0000, A 0.000, B 0.000, C 0.000 }
gfCNCPoint6[6619] = {X 170.0416, Y 39.6939, Z -8.0000, A 0.000, B 0.000, C 0.000 }
gfCNCPoint6[6620] = {X 169.6860, Y 38.2306, Z -8.0000, A 0.000, B 0.000, C 0.000 }
gfCNCPoint6[6621] = {X 169.6310, Y 37.8853, Z -8.0000, A 0.000, B 0.000, C 0.000 }
gfCNCPoint6[6622] = {X 165.6018, Y 38.5269, Z -8.0000, A 0.000, B 0.000, C 0.000 }
gfCNCPoint6[6623] = {X 165.6018, Y 38.5269, Z -5.0000, A 0.000, B 0.000, C 0.000 }
gfCNCPoint6[6624] = {X 165.6018, Y 38.5269, Z 11.0000, A 0.000, B 0.000, C 0.000 }
gfCNCPoint6[6625] = {X 210.1635, Y 28.5736, Z 11.0000, A 0.000, B 0.000, C 0.000 }
gfCNCPoint6[6626] = {X 210.1635, Y 28.5736, Z -5.0000, A 0.000, B 0.000, C 0.000 }
gfCNCPoint6[6627] = {X 210.1635, Y 28.5736, Z -8.0000, A 0.000, B 0.000, C 0.000 }
gfCNCPoint6[6628] = {X 214.2435, Y 28.5736, Z -8.0000, A 0.000, B 0.000, C 0.000 }
gfCNCPoint6[6629] = {X 214.2435, Y 17.4625, Z -8.0000, A 0.000, B 0.000, C 0.000 }
gfCNCPoint6[6630] = {X 214.2382, Y 16.7691, Z -8.0000, A 0.000, B 0.000, C 0.000 }
gfCNCPoint6[6631] = {X 214.2418, Y 16.2718, Z -8.0000, A 0.000, B 0.000, C 0.000 }
gfCNCPoint6[6632] = {X 213.6043, Y 15.6008, Z -8.0000, A 0.000, B 0.000, C 0.000 }
gfCNCPoint6[6633] = {X 213.1244, Y 14.8093, Z -8.0000, A 0.000, B 0.000, C 0.000 }
gfCNCPoint6[6634] = {X 212.8241, Y 13.9337, Z -8.0000, A 0.000, B 0.000, C 0.000 }
gfCNCPoint6[6635] = {X 212.7172, Y 13.0143, Z -8.0000, A 0.000, B 0.000, C 0.000 }
gfCNCPoint6[6636] = {X 212.7170, Y 12.1868, Z -8.0000, A 0.000, B 0.000, C 0.000 }
gfCNCPoint6[6637] = {X 212.8253, Y 11.2255, Z -8.0000, A 0.000, B 0.000, C 0.000 }
gfCNCPoint6[6638] = {X 213.1448, Y 10.3124, Z -8.0000, A 0.000, B 0.000, C 0.000 }
gfCNCPoint6[6639] = {X 213.6595, Y 9.4933, Z -8.0000, A 0.000, B 0.000, C 0.000 }
gfCNCPoint6[6640] = {X 214.3435, Y 8.8093, Z -8.0000, A 0.000, B 0.000, C 0.000 }
gfCNCPoint6[6641] = {X 215.1626, Y 8.2946, Z -8.0000, A 0.000, B 0.000, C 0.000 }
gfCNCPoint6[6642] = {X 216.0757, Y 7.9751, Z -8.0000, A 0.000, B 0.000, C 0.000 }
gfCNCPoint6[6643] = {X 217.0370, Y 7.8668, Z -8.0000, A 0.000, B 0.000, C 0.000 }
gfCNCPoint6[6644] = {X 223.4805, Y 7.8668, Z -8.0000, A 0.000, B 0.000, C 0.000 }
gfCNCPoint6[6645] = {X 224.4418, Y 7.9751, Z -8.0000, A 0.000, B 0.000, C 0.000 }
gfCNCPoint6[6646] = {X 225.3549, Y 8.2946, Z -8.0000, A 0.000, B 0.000, C 0.000 }
gfCNCPoint6[6647] = {X 226.1740, Y 8.8093, Z -8.0000, A 0.000, B 0.000, C 0.000 }
gfCNCPoint6[6648] = {X 226.8580, Y 9.4933, Z -8.0000, A 0.000, B 0.000, C 0.000 }
gfCNCPoint6[6649] = {X 227.3727, Y 10.3124, Z -8.0000, A 0.000, B 0.000, C 0.000 }
gfCNCPoint6[6650] = {X 227.6922, Y 11.2255, Z -8.0000, A 0.000, B 0.000, C 0.000 }
gfCNCPoint6[6651] = {X 227.8005, Y 12.1868, Z -8.0000, A 0.000, B 0.000, C 0.000 }
gfCNCPoint6[6652] = {X 227.8005, Y 12.9782, Z -8.0000, A 0.000, B 0.000, C 0.000 }
gfCNCPoint6[6653] = {X 227.6992, Y 13.9078, Z -8.0000, A 0.000, B 0.000, C 0.000 }
gfCNCPoint6[6654] = {X 227.4003, Y 14.7938, Z -8.0000, A 0.000, B 0.000, C 0.000 }
gfCNCPoint6[6655] = {X 226.9178, Y 15.5948, Z -8.0000, A 0.000, B 0.000, C 0.000 }
gfCNCPoint6[6656] = {X 226.2742, Y 16.2731, Z -8.0000, A 0.000, B 0.000, C 0.000 }
gfCNCPoint6[6657] = {X 226.2754, Y 40.9157, Z -8.0000, A 0.000, B 0.000, C 0.000 }
gfCNCPoint6[6658] = {X 226.9123, Y 41.5858, Z -8.0000, A 0.000, B 0.000, C 0.000 }
gfCNCPoint6[6659] = {X 227.3921, Y 42.3762, Z -8.0000, A 0.000, B 0.000, C 0.000 }
gfCNCPoint6[6660] = {X 227.6927, Y 43.2506, Z -8.0000, A 0.000, B 0.000, C 0.000 }
gfCNCPoint6[6661] = {X 227.8003, Y 44.1689, Z -8.0000, A 0.000, B 0.000, C 0.000 }
gfCNCPoint6[6662] = {X 227.8005, Y 45.0000, Z -8.0000, A 0.000, B 0.000, C 0.000 }
gfCNCPoint6[6663] = {X 227.6922, Y 45.9613, Z -8.0000, A 0.000, B 0.000, C 0.000 }
gfCNCPoint6[6664] = {X 227.3727, Y 46.8744, Z -8.0000, A 0.000, B 0.000, C 0.000 }
gfCNCPoint6[6665] = {X 226.8580, Y 47.6935, Z -8.0000, A 0.000, B 0.000, C 0.000 }
gfCNCPoint6[6666] = {X 226.1740, Y 48.3775, Z -8.0000, A 0.000, B 0.000, C 0.000 }
gfCNCPoint6[6667] = {X 225.3549, Y 48.8922, Z -8.0000, A 0.000, B 0.000, C 0.000 }
gfCNCPoint6[6668] = {X 224.4418, Y 49.2117, Z -8.0000, A 0.000, B 0.000, C 0.000 }
gfCNCPoint6[6669] = {X 223.4805, Y 49.3200, Z -8.0000, A 0.000, B 0.000, C 0.000 }
gfCNCPoint6[6670] = {X 217.0370, Y 49.3200, Z -8.0000, A 0.000, B 0.000, C 0.000 }
gfCNCPoint6[6671] = {X 216.0805, Y 49.2128, Z -8.0000, A 0.000, B 0.000, C 0.000 }
gfCNCPoint6[6672] = {X 215.1715, Y 48.8964, Z -8.0000, A 0.000, B 0.000, C 0.000 }
gfCNCPoint6[6673] = {X 214.3551, Y 48.3867, Z -8.0000, A 0.000, B 0.000, C 0.000 }
gfCNCPoint6[6674] = {X 213.6718, Y 47.7088, Z -8.0000, A 0.000, B 0.000, C 0.000 }
gfCNCPoint6[6675] = {X 213.1556, Y 46.8965, Z -8.0000, A 0.000, B 0.000, C 0.000 }
gfCNCPoint6[6676] = {X 212.8320, Y 45.9901, Z -8.0000, A 0.000, B 0.000, C 0.000 }
gfCNCPoint6[6677] = {X 212.7172, Y 45.0345, Z -8.0000, A 0.000, B 0.000, C 0.000 }
gfCNCPoint6[6678] = {X 212.7170, Y 44.1900, Z -8.0000, A 0.000, B 0.000, C 0.000 }
gfCNCPoint6[6679] = {X 212.7887, Y 43.4139, Z -8.0000, A 0.000, B 0.000, C 0.000 }
gfCNCPoint6[6680] = {X 213.0012, Y 42.6640, Z -8.0000, A 0.000, B 0.000, C 0.000 }
gfCNCPoint6[6681] = {X 213.3474, Y 41.9657, Z -8.0000, A 0.000, B 0.000, C 0.000 }
gfCNCPoint6[6682] = {X 213.8156, Y 41.3425, Z -8.0000, A 0.000, B 0.000, C 0.000 }
gfCNCPoint6[6683] = {X 214.2392, Y 40.8754, Z -8.0000, A 0.000, B 0.000, C 0.000 }
gfCNCPoint6[6684] = {X 214.2435, Y 40.3061, Z -8.0000, A 0.000, B 0.000, C 0.000 }
gfCNCPoint6[6685] = {X 214.2435, Y 28.5736, Z -8.0000, A 0.000, B 0.000, C 0.000 }
gfCNCPoint6[6686] = {X 210.2435, Y 28.5736, Z -8.0000, A 0.000, B 0.000, C 0.000 }
gfCNCPoint6[6687] = {X 214.3235, Y 28.5736, Z -8.0000, A 0.000, B 0.000, C 0.000 }
gfCNCPoint6[6688] = {X 214.3235, Y 17.4621, Z -8.0000, A 0.000, B 0.000, C 0.000 }
gfCNCPoint6[6689] = {X 214.3182, Y 16.7691, Z -8.0000, A 0.000, B 0.000, C 0.000 }
gfCNCPoint6[6690] = {X 214.3221, Y 16.2348, Z -8.0000, A 0.000, B 0.000, C 0.000 }
gfCNCPoint6[6691] = {X 213.6849, Y 15.5743, Z -8.0000, A 0.000, B 0.000, C 0.000 }
gfCNCPoint6[6692] = {X 213.2048, Y 14.7922, Z -8.0000, A 0.000, B 0.000, C 0.000 }
gfCNCPoint6[6693] = {X 212.9041, Y 13.9251, Z -8.0000, A 0.000, B 0.000, C 0.000 }
gfCNCPoint6[6694] = {X 212.7972, Y 13.0137, Z -8.0000, A 0.000, B 0.000, C 0.000 }
gfCNCPoint6[6695] = {X 212.7970, Y 12.1868, Z -8.0000, A 0.000, B 0.000, C 0.000 }
gfCNCPoint6[6696] = {X 212.9033, Y 11.2433, Z -8.0000, A 0.000, B 0.000, C 0.000 }
gfCNCPoint6[6697] = {X 213.2169, Y 10.3472, Z -8.0000, A 0.000, B 0.000, C 0.000 }
gfCNCPoint6[6698] = {X 213.7220, Y 9.5432, Z -8.0000, A 0.000, B 0.000, C 0.000 }
gfCNCPoint6[6699] = {X 214.3934, Y 8.8719, Z -8.0000, A 0.000, B 0.000, C 0.000 }
gfCNCPoint6[6700] = {X 215.1973, Y 8.3667, Z -8.0000, A 0.000, B 0.000, C 0.000 }
gfCNCPoint6[6701] = {X 216.0935, Y 8.0531, Z -8.0000, A 0.000, B 0.000, C 0.000 }
gfCNCPoint6[6702] = {X 217.0370, Y 7.9468, Z -8.0000, A 0.000, B 0.000, C 0.000 }
gfCNCPoint6[6703] = {X 223.4805, Y 7.9468, Z -8.0000, A 0.000, B 0.000, C 0.000 }
gfCNCPoint6[6704] = {X 224.4240, Y 8.0531, Z -8.0000, A 0.000, B 0.000, C 0.000 }
gfCNCPoint6[6705] = {X 225.3201, Y 8.3667, Z -8.0000, A 0.000, B 0.000, C 0.000 }
gfCNCPoint6[6706] = {X 226.1241, Y 8.8718, Z -8.0000, A 0.000, B 0.000, C 0.000 }
gfCNCPoint6[6707] = {X 226.7954, Y 9.5432, Z -8.0000, A 0.000, B 0.000, C 0.000 }
gfCNCPoint6[6708] = {X 227.3006, Y 10.3471, Z -8.0000, A 0.000, B 0.000, C 0.000 }
gfCNCPoint6[6709] = {X 227.6142, Y 11.2433, Z -8.0000, A 0.000, B 0.000, C 0.000 }
gfCNCPoint6[6710] = {X 227.7205, Y 12.1868, Z -8.0000, A 0.000, B 0.000, C 0.000 }
gfCNCPoint6[6711] = {X 227.7205, Y 12.9782, Z -8.0000, A 0.000, B 0.000, C 0.000 }
gfCNCPoint6[6712] = {X 227.6191, Y 13.8996, Z -8.0000, A 0.000, B 0.000, C 0.000 }
gfCNCPoint6[6713] = {X 227.3200, Y 14.7769, Z -8.0000, A 0.000, B 0.000, C 0.000 }
gfCNCPoint6[6714] = {X 226.8373, Y 15.5683, Z -8.0000, A 0.000, B 0.000, C 0.000 }
gfCNCPoint6[6715] = {X 226.1942, Y 16.2359, Z -8.0000, A 0.000, B 0.000, C 0.000 }
gfCNCPoint6[6716] = {X 226.1954, Y 40.9529, Z -8.0000, A 0.000, B 0.000, C 0.000 }
gfCNCPoint6[6717] = {X 226.8319, Y 41.6125, Z -8.0000, A 0.000, B 0.000, C 0.000 }
gfCNCPoint6[6718] = {X 227.3118, Y 42.3935, Z -8.0000, A 0.000, B 0.000, C 0.000 }
gfCNCPoint6[6719] = {X 227.6126, Y 43.2594, Z -8.0000, A 0.000, B 0.000, C 0.000 }
gfCNCPoint6[6720] = {X 227.7203, Y 44.1697, Z -8.0000, A 0.000, B 0.000, C 0.000 }
gfCNCPoint6[6721] = {X 227.7205, Y 45.0000, Z -8.0000, A 0.000, B 0.000, C 0.000 }
gfCNCPoint6[6722] = {X 227.6142, Y 45.9435, Z -8.0000, A 0.000, B 0.000, C 0.000 }
gfCNCPoint6[6723] = {X 227.3006, Y 46.8397, Z -8.0000, A 0.000, B 0.000, C 0.000 }
gfCNCPoint6[6724] = {X 226.7954, Y 47.6436, Z -8.0000, A 0.000, B 0.000, C 0.000 }
gfCNCPoint6[6725] = {X 226.1241, Y 48.3150, Z -8.0000, A 0.000, B 0.000, C 0.000 }
gfCNCPoint6[6726] = {X 225.3201, Y 48.8201, Z -8.0000, A 0.000, B 0.000, C 0.000 }
gfCNCPoint6[6727] = {X 224.4240, Y 49.1337, Z -8.0000, A 0.000, B 0.000, C 0.000 }
gfCNCPoint6[6728] = {X 223.4805, Y 49.2400, Z -8.0000, A 0.000, B 0.000, C 0.000 }
gfCNCPoint6[6729] = {X 217.0370, Y 49.2400, Z -8.0000, A 0.000, B 0.000, C 0.000 }
gfCNCPoint6[6730] = {X 216.0982, Y 49.1348, Z -8.0000, A 0.000, B 0.000, C 0.000 }
gfCNCPoint6[6731] = {X 215.2061, Y 48.8243, Z -8.0000, A 0.000, B 0.000, C 0.000 }
gfCNCPoint6[6732] = {X 214.4048, Y 48.3240, Z -8.0000, A 0.000, B 0.000, C 0.000 }
gfCNCPoint6[6733] = {X 213.7341, Y 47.6587, Z -8.0000, A 0.000, B 0.000, C 0.000 }
gfCNCPoint6[6734] = {X 213.2275, Y 46.8614, Z -8.0000, A 0.000, B 0.000, C 0.000 }
gfCNCPoint6[6735] = {X 212.9099, Y 45.9717, Z -8.0000, A 0.000, B 0.000, C 0.000 }
gfCNCPoint6[6736] = {X 212.7972, Y 45.0338, Z -8.0000, A 0.000, B 0.000, C 0.000 }
gfCNCPoint6[6737] = {X 212.7970, Y 44.1900, Z -8.0000, A 0.000, B 0.000, C 0.000 }
gfCNCPoint6[6738] = {X 212.8673, Y 43.4285, Z -8.0000, A 0.000, B 0.000, C 0.000 }
gfCNCPoint6[6739] = {X 213.0758, Y 42.6928, Z -8.0000, A 0.000, B 0.000, C 0.000 }
gfCNCPoint6[6740] = {X 213.4155, Y 42.0076, Z -8.0000, A 0.000, B 0.000, C 0.000 }
gfCNCPoint6[6741] = {X 213.8749, Y 41.3962, Z -8.0000, A 0.000, B 0.000, C 0.000 }
gfCNCPoint6[6742] = {X 214.3189, Y 40.9065, Z -8.0000, A 0.000, B 0.000, C 0.000 }
gfCNCPoint6[6743] = {X 214.3235, Y 40.3065, Z -8.0000, A 0.000, B 0.000, C 0.000 }
gfCNCPoint6[6744] = {X 214.3235, Y 28.5736, Z -8.0000, A 0.000, B 0.000, C 0.000 }
gfCNCPoint6[6745] = {X 210.3235, Y 28.5736, Z -8.0000, A 0.000, B 0.000, C 0.000 }
gfCNCPoint6[6746] = {X 214.4035, Y 28.5736, Z -8.0000, A 0.000, B 0.000, C 0.000 }
gfCNCPoint6[6747] = {X 214.4035, Y 17.4618, Z -8.0000, A 0.000, B 0.000, C 0.000 }
gfCNCPoint6[6748] = {X 214.3982, Y 16.7691, Z -8.0000, A 0.000, B 0.000, C 0.000 }
gfCNCPoint6[6749] = {X 214.4023, Y 16.1974, Z -8.0000, A 0.000, B 0.000, C 0.000 }
gfCNCPoint6[6750] = {X 213.7655, Y 15.5476, Z -8.0000, A 0.000, B 0.000, C 0.000 }
gfCNCPoint6[6751] = {X 213.2852, Y 14.7750, Z -8.0000, A 0.000, B 0.000, C 0.000 }
gfCNCPoint6[6752] = {X 212.9842, Y 13.9164, Z -8.0000, A 0.000, B 0.000, C 0.000 }
gfCNCPoint6[6753] = {X 212.8772, Y 13.0130, Z -8.0000, A 0.000, B 0.000, C 0.000 }
gfCNCPoint6[6754] = {X 212.8770, Y 12.1868, Z -8.0000, A 0.000, B 0.000, C 0.000 }
gfCNCPoint6[6755] = {X 212.9813, Y 11.2611, Z -8.0000, A 0.000, B 0.000, C 0.000 }
gfCNCPoint6[6756] = {X 213.2890, Y 10.3819, Z -8.0000, A 0.000, B 0.000, C 0.000 }
gfCNCPoint6[6757] = {X 213.7846, Y 9.5931, Z -8.0000, A 0.000, B 0.000, C 0.000 }
gfCNCPoint6[6758] = {X 214.4433, Y 8.9344, Z -8.0000, A 0.000, B 0.000, C 0.000 }
gfCNCPoint6[6759] = {X 215.2321, Y 8.4388, Z -8.0000, A 0.000, B 0.000, C 0.000 }
gfCNCPoint6[6760] = {X 216.1113, Y 8.1311, Z -8.0000, A 0.000, B 0.000, C 0.000 }
gfCNCPoint6[6761] = {X 217.0370, Y 8.0268, Z -8.0000, A 0.000, B 0.000, C 0.000 }
gfCNCPoint6[6762] = {X 223.4805, Y 8.0268, Z -8.0000, A 0.000, B 0.000, C 0.000 }
gfCNCPoint6[6763] = {X 224.4062, Y 8.1311, Z -8.0000, A 0.000, B 0.000, C 0.000 }
gfCNCPoint6[6764] = {X 225.2854, Y 8.4388, Z -8.0000, A 0.000, B 0.000, C 0.000 }
gfCNCPoint6[6765] = {X 226.0742, Y 8.9344, Z -8.0000, A 0.000, B 0.000, C 0.000 }
gfCNCPoint6[6766] = {X 226.7329, Y 9.5931, Z -8.0000, A 0.000, B 0.000, C 0.000 }
gfCNCPoint6[6767] = {X 227.2285, Y 10.3819, Z -8.0000, A 0.000, B 0.000, C 0.000 }
gfCNCPoint6[6768] = {X 227.5362, Y 11.2611, Z -8.0000, A 0.000, B 0.000, C 0.000 }
gfCNCPoint6[6769] = {X 227.6405, Y 12.1868, Z -8.0000, A 0.000, B 0.000, C 0.000 }
gfCNCPoint6[6770] = {X 227.6405, Y 12.9782, Z -8.0000, A 0.000, B 0.000, C 0.000 }
gfCNCPoint6[6771] = {X 227.5390, Y 13.8913, Z -8.0000, A 0.000, B 0.000, C 0.000 }
gfCNCPoint6[6772] = {X 227.2396, Y 14.7599, Z -8.0000, A 0.000, B 0.000, C 0.000 }
gfCNCPoint6[6773] = {X 226.7568, Y 15.5415, Z -8.0000, A 0.000, B 0.000, C 0.000 }
gfCNCPoint6[6774] = {X 226.1142, Y 16.1982, Z -8.0000, A 0.000, B 0.000, C 0.000 }
gfCNCPoint6[6775] = {X 226.1154, Y 40.9906, Z -8.0000, A 0.000, B 0.000, C 0.000 }
gfCNCPoint6[6776] = {X 226.7515, Y 41.6394, Z -8.0000, A 0.000, B 0.000, C 0.000 }
gfCNCPoint6[6777] = {X 227.2315, Y 42.4109, Z -8.0000, A 0.000, B 0.000, C 0.000 }
gfCNCPoint6[6778] = {X 227.5325, Y 43.2682, Z -8.0000, A 0.000, B 0.000, C 0.000 }
gfCNCPoint6[6779] = {X 227.6403, Y 44.1704, Z -8.0000, A 0.000, B 0.000, C 0.000 }
gfCNCPoint6[6780] = {X 227.6405, Y 45.0000, Z -8.0000, A 0.000, B 0.000, C 0.000 }
gfCNCPoint6[6781] = {X 227.5362, Y 45.9257, Z -8.0000, A 0.000, B 0.000, C 0.000 }
gfCNCPoint6[6782] = {X 227.2285, Y 46.8050, Z -8.0000, A 0.000, B 0.000, C 0.000 }
gfCNCPoint6[6783] = {X 226.7329, Y 47.5937, Z -8.0000, A 0.000, B 0.000, C 0.000 }
gfCNCPoint6[6784] = {X 226.0742, Y 48.2524, Z -8.0000, A 0.000, B 0.000, C 0.000 }
gfCNCPoint6[6785] = {X 225.2854, Y 48.7480, Z -8.0000, A 0.000, B 0.000, C 0.000 }
gfCNCPoint6[6786] = {X 224.4062, Y 49.0557, Z -8.0000, A 0.000, B 0.000, C 0.000 }
gfCNCPoint6[6787] = {X 223.4805, Y 49.1600, Z -8.0000, A 0.000, B 0.000, C 0.000 }
gfCNCPoint6[6788] = {X 217.0370, Y 49.1600, Z -8.0000, A 0.000, B 0.000, C 0.000 }
gfCNCPoint6[6789] = {X 216.1160, Y 49.0568, Z -8.0000, A 0.000, B 0.000, C 0.000 }
gfCNCPoint6[6790] = {X 215.2406, Y 48.7521, Z -8.0000, A 0.000, B 0.000, C 0.000 }
gfCNCPoint6[6791] = {X 214.4544, Y 48.2613, Z -8.0000, A 0.000, B 0.000, C 0.000 }
gfCNCPoint6[6792] = {X 213.7965, Y 47.6085, Z -8.0000, A 0.000, B 0.000, C 0.000 }
gfCNCPoint6[6793] = {X 213.2993, Y 46.8263, Z -8.0000, A 0.000, B 0.000, C 0.000 }
gfCNCPoint6[6794] = {X 212.9877, Y 45.9534, Z -8.0000, A 0.000, B 0.000, C 0.000 }
gfCNCPoint6[6795] = {X 212.8771, Y 45.0332, Z -8.0000, A 0.000, B 0.000, C 0.000 }
gfCNCPoint6[6796] = {X 212.8770, Y 44.1900, Z -8.0000, A 0.000, B 0.000, C 0.000 }
gfCNCPoint6[6797] = {X 212.9460, Y 43.4432, Z -8.0000, A 0.000, B 0.000, C 0.000 }
gfCNCPoint6[6798] = {X 213.1505, Y 42.7216, Z -8.0000, A 0.000, B 0.000, C 0.000 }
gfCNCPoint6[6799] = {X 213.4836, Y 42.0496, Z -8.0000, A 0.000, B 0.000, C 0.000 }
gfCNCPoint6[6800] = {X 213.9342, Y 41.4500, Z -8.0000, A 0.000, B 0.000, C 0.000 }
gfCNCPoint6[6801] = {X 214.3987, Y 40.9376, Z -8.0000, A 0.000, B 0.000, C 0.000 }
gfCNCPoint6[6802] = {X 214.4035, Y 40.3068, Z -8.0000, A 0.000, B 0.000, C 0.000 }
gfCNCPoint6[6803] = {X 214.4035, Y 28.5736, Z -8.0000, A 0.000, B 0.000, C 0.000 }
gfCNCPoint6[6804] = {X 210.4035, Y 28.5736, Z -8.0000, A 0.000, B 0.000, C 0.000 }
gfCNCPoint6[6805] = {X 214.4835, Y 28.5736, Z -8.0000, A 0.000, B 0.000, C 0.000 }
gfCNCPoint6[6806] = {X 214.4835, Y 17.4614, Z -8.0000, A 0.000, B 0.000, C 0.000 }
gfCNCPoint6[6807] = {X 214.4782, Y 16.7691, Z -8.0000, A 0.000, B 0.000, C 0.000 }
gfCNCPoint6[6808] = {X 214.4826, Y 16.1594, Z -8.0000, A 0.000, B 0.000, C 0.000 }
gfCNCPoint6[6809] = {X 214.4245, Y 16.1119, Z -8.0000, A 0.000, B 0.000, C 0.000 }
gfCNCPoint6[6810] = {X 214.3672, Y 16.0632, Z -8.0000, A 0.000, B 0.000, C 0.000 }
gfCNCPoint6[6811] = {X 213.7772, Y 15.4315, Z -8.0000, A 0.000, B 0.000, C 0.000 }
gfCNCPoint6[6812] = {X 213.3334, Y 14.6897, Z -8.0000, A 0.000, B 0.000, C 0.000 }
gfCNCPoint6[6813] = {X 213.0559, Y 13.8711, Z -8.0000, A 0.000, B 0.000, C 0.000 }
gfCNCPoint6[6814] = {X 212.9572, Y 13.0123, Z -8.0000, A 0.000, B 0.000, C 0.000 }
gfCNCPoint6[6815] = {X 212.9570, Y 12.1868, Z -8.0000, A 0.000, B 0.000, C 0.000 }
gfCNCPoint6[6816] = {X 213.0593, Y 11.2789, Z -8.0000, A 0.000, B 0.000, C 0.000 }
gfCNCPoint6[6817] = {X 213.3611, Y 10.4166, Z -8.0000, A 0.000, B 0.000, C 0.000 }
gfCNCPoint6[6818] = {X 213.8471, Y 9.6430, Z -8.0000, A 0.000, B 0.000, C 0.000 }
gfCNCPoint6[6819] = {X 214.4932, Y 8.9969, Z -8.0000, A 0.000, B 0.000, C 0.000 }
gfCNCPoint6[6820] = {X 215.2668, Y 8.5109, Z -8.0000, A 0.000, B 0.000, C 0.000 }
gfCNCPoint6[6821] = {X 216.1291, Y 8.2091, Z -8.0000, A 0.000, B 0.000, C 0.000 }
gfCNCPoint6[6822] = {X 217.0370, Y 8.1068, Z -8.0000, A 0.000, B 0.000, C 0.000 }
gfCNCPoint6[6823] = {X 223.4805, Y 8.1068, Z -8.0000, A 0.000, B 0.000, C 0.000 }
gfCNCPoint6[6824] = {X 224.3884, Y 8.2091, Z -8.0000, A 0.000, B 0.000, C 0.000 }
gfCNCPoint6[6825] = {X 225.2507, Y 8.5109, Z -8.0000, A 0.000, B 0.000, C 0.000 }
gfCNCPoint6[6826] = {X 226.0243, Y 8.9969, Z -8.0000, A 0.000, B 0.000, C 0.000 }
gfCNCPoint6[6827] = {X 226.6704, Y 9.6430, Z -8.0000, A 0.000, B 0.000, C 0.000 }
gfCNCPoint6[6828] = {X 227.1564, Y 10.4166, Z -8.0000, A 0.000, B 0.000, C 0.000 }
gfCNCPoint6[6829] = {X 227.4582, Y 11.2789, Z -8.0000, A 0.000, B 0.000, C 0.000 }
gfCNCPoint6[6830] = {X 227.5605, Y 12.1868, Z -8.0000, A 0.000, B 0.000, C 0.000 }
gfCNCPoint6[6831] = {X 227.5605, Y 12.9782, Z -8.0000, A 0.000, B 0.000, C 0.000 }
gfCNCPoint6[6832] = {X 227.4589, Y 13.8829, Z -8.0000, A 0.000, B 0.000, C 0.000 }
gfCNCPoint6[6833] = {X 227.1591, Y 14.7427, Z -8.0000, A 0.000, B 0.000, C 0.000 }
gfCNCPoint6[6834] = {X 226.6762, Y 15.5145, Z -8.0000, A 0.000, B 0.000, C 0.000 }
gfCNCPoint6[6835] = {X 226.0342, Y 16.1600, Z -8.0000, A 0.000, B 0.000, C 0.000 }
gfCNCPoint6[6836] = {X 226.0354, Y 41.0282, Z -8.0000, A 0.000, B 0.000, C 0.000 }
gfCNCPoint6[6837] = {X 226.1412, Y 41.1158, Z -8.0000, A 0.000, B 0.000, C 0.000 }
gfCNCPoint6[6838] = {X 226.7344, Y 41.7474, Z -8.0000, A 0.000, B 0.000, C 0.000 }
gfCNCPoint6[6839] = {X 227.1808, Y 42.4902, Z -8.0000, A 0.000, B 0.000, C 0.000 }
gfCNCPoint6[6840] = {X 227.4603, Y 43.3104, Z -8.0000, A 0.000, B 0.000, C 0.000 }
gfCNCPoint6[6841] = {X 227.5603, Y 44.1712, Z -8.0000, A 0.000, B 0.000, C 0.000 }
gfCNCPoint6[6842] = {X 227.5605, Y 45.0000, Z -8.0000, A 0.000, B 0.000, C 0.000 }
gfCNCPoint6[6843] = {X 227.4582, Y 45.9079, Z -8.0000, A 0.000, B 0.000, C 0.000 }
gfCNCPoint6[6844] = {X 227.1564, Y 46.7702, Z -8.0000, A 0.000, B 0.000, C 0.000 }
gfCNCPoint6[6845] = {X 226.6704, Y 47.5438, Z -8.0000, A 0.000, B 0.000, C 0.000 }
gfCNCPoint6[6846] = {X 226.0243, Y 48.1899, Z -8.0000, A 0.000, B 0.000, C 0.000 }
gfCNCPoint6[6847] = {X 225.2507, Y 48.6760, Z -8.0000, A 0.000, B 0.000, C 0.000 }
gfCNCPoint6[6848] = {X 224.3884, Y 48.9777, Z -8.0000, A 0.000, B 0.000, C 0.000 }
gfCNCPoint6[6849] = {X 223.4805, Y 49.0800, Z -8.0000, A 0.000, B 0.000, C 0.000 }
gfCNCPoint6[6850] = {X 217.0370, Y 49.0800, Z -8.0000, A 0.000, B 0.000, C 0.000 }
gfCNCPoint6[6851] = {X 216.1337, Y 48.9787, Z -8.0000, A 0.000, B 0.000, C 0.000 }
gfCNCPoint6[6852] = {X 215.2752, Y 48.6800, Z -8.0000, A 0.000, B 0.000, C 0.000 }
gfCNCPoint6[6853] = {X 214.5041, Y 48.1986, Z -8.0000, A 0.000, B 0.000, C 0.000 }
gfCNCPoint6[6854] = {X 213.8588, Y 47.5584, Z -8.0000, A 0.000, B 0.000, C 0.000 }
gfCNCPoint6[6855] = {X 213.3712, Y 46.7912, Z -8.0000, A 0.000, B 0.000, C 0.000 }
gfCNCPoint6[6856] = {X 213.0656, Y 45.9351, Z -8.0000, A 0.000, B 0.000, C 0.000 }
gfCNCPoint6[6857] = {X 212.9571, Y 45.0325, Z -8.0000, A 0.000, B 0.000, C 0.000 }
gfCNCPoint6[6858] = {X 212.9570, Y 44.1900, Z -8.0000, A 0.000, B 0.000, C 0.000 }
gfCNCPoint6[6859] = {X 213.0246, Y 43.4578, Z -8.0000, A 0.000, B 0.000, C 0.000 }
gfCNCPoint6[6860] = {X 213.2251, Y 42.7504, Z -8.0000, A 0.000, B 0.000, C 0.000 }
gfCNCPoint6[6861] = {X 213.5517, Y 42.0916, Z -8.0000, A 0.000, B 0.000, C 0.000 }
gfCNCPoint6[6862] = {X 213.9934, Y 41.5037, Z -8.0000, A 0.000, B 0.000, C 0.000 }
gfCNCPoint6[6863] = {X 214.4784, Y 40.9687, Z -8.0000, A 0.000, B 0.000, C 0.000 }
gfCNCPoint6[6864] = {X 214.4835, Y 40.3072, Z -8.0000, A 0.000, B 0.000, C 0.000 }
gfCNCPoint6[6865] = {X 214.4835, Y 28.5736, Z -8.0000, A 0.000, B 0.000, C 0.000 }
gfCNCPoint6[6866] = {X 210.4835, Y 28.5736, Z -8.0000, A 0.000, B 0.000, C 0.000 }
gfCNCPoint6[6867] = {X 214.5635, Y 28.5736, Z -8.0000, A 0.000, B 0.000, C 0.000 }
gfCNCPoint6[6868] = {X 214.5635, Y 17.4611, Z -8.0000, A 0.000, B 0.000, C 0.000 }
gfCNCPoint6[6869] = {X 214.5582, Y 16.7687, Z -8.0000, A 0.000, B 0.000, C 0.000 }
gfCNCPoint6[6870] = {X 214.5577, Y 16.1872, Z -8.0000, A 0.000, B 0.000, C 0.000 }
gfCNCPoint6[6871] = {X 214.5756, Y 16.1310, Z -8.0000, A 0.000, B 0.000, C 0.000 }
gfCNCPoint6[6872] = {X 214.4968, Y 16.0679, Z -8.0000, A 0.000, B 0.000, C 0.000 }
gfCNCPoint6[6873] = {X 214.4196, Y 16.0028, Z -8.0000, A 0.000, B 0.000, C 0.000 }
gfCNCPoint6[6874] = {X 213.8360, Y 15.3767, Z -8.0000, A 0.000, B 0.000, C 0.000 }
gfCNCPoint6[6875] = {X 213.3990, Y 14.6409, Z -8.0000, A 0.000, B 0.000, C 0.000 }
gfCNCPoint6[6876] = {X 213.1286, Y 13.8289, Z -8.0000, A 0.000, B 0.000, C 0.000 }
gfCNCPoint6[6877] = {X 213.0370, Y 12.9780, Z -8.0000, A 0.000, B 0.000, C 0.000 }
gfCNCPoint6[6878] = {X 213.0370, Y 12.1868, Z -8.0000, A 0.000, B 0.000, C 0.000 }
gfCNCPoint6[6879] = {X 213.1373, Y 11.2967, Z -8.0000, A 0.000, B 0.000, C 0.000 }
gfCNCPoint6[6880] = {X 213.4331, Y 10.4513, Z -8.0000, A 0.000, B 0.000, C 0.000 }
gfCNCPoint6[6881] = {X 213.9097, Y 9.6929, Z -8.0000, A 0.000, B 0.000, C 0.000 }
gfCNCPoint6[6882] = {X 214.5431, Y 9.0595, Z -8.0000, A 0.000, B 0.000, C 0.000 }
gfCNCPoint6[6883] = {X 215.3015, Y 8.5829, Z -8.0000, A 0.000, B 0.000, C 0.000 }
gfCNCPoint6[6884] = {X 216.1469, Y 8.2871, Z -8.0000, A 0.000, B 0.000, C 0.000 }
gfCNCPoint6[6885] = {X 217.0370, Y 8.1868, Z -8.0000, A 0.000, B 0.000, C 0.000 }
gfCNCPoint6[6886] = {X 223.4805, Y 8.1868, Z -8.0000, A 0.000, B 0.000, C 0.000 }
gfCNCPoint6[6887] = {X 224.3706, Y 8.2871, Z -8.0000, A 0.000, B 0.000, C 0.000 }
gfCNCPoint6[6888] = {X 225.2160, Y 8.5829, Z -8.0000, A 0.000, B 0.000, C 0.000 }
gfCNCPoint6[6889] = {X 225.9744, Y 9.0595, Z -8.0000, A 0.000, B 0.000, C 0.000 }
gfCNCPoint6[6890] = {X 226.6078, Y 9.6929, Z -8.0000, A 0.000, B 0.000, C 0.000 }
gfCNCPoint6[6891] = {X 227.0844, Y 10.4513, Z -8.0000, A 0.000, B 0.000, C 0.000 }
gfCNCPoint6[6892] = {X 227.3802, Y 11.2967, Z -8.0000, A 0.000, B 0.000, C 0.000 }
gfCNCPoint6[6893] = {X 227.4805, Y 12.1868, Z -8.0000, A 0.000, B 0.000, C 0.000 }
gfCNCPoint6[6894] = {X 227.4803, Y 13.0192, Z -8.0000, A 0.000, B 0.000, C 0.000 }
gfCNCPoint6[6895] = {X 227.3717, Y 13.9045, Z -8.0000, A 0.000, B 0.000, C 0.000 }
gfCNCPoint6[6896] = {X 227.0697, Y 14.7437, Z -8.0000, A 0.000, B 0.000, C 0.000 }
gfCNCPoint6[6897] = {X 226.5892, Y 15.4951, Z -8.0000, A 0.000, B 0.000, C 0.000 }
gfCNCPoint6[6898] = {X 225.9542, Y 16.1214, Z -8.0000, A 0.000, B 0.000, C 0.000 }
gfCNCPoint6[6899] = {X 225.9554, Y 41.0659, Z -8.0000, A 0.000, B 0.000, C 0.000 }
gfCNCPoint6[6900] = {X 226.0940, Y 41.1807, Z -8.0000, A 0.000, B 0.000, C 0.000 }
gfCNCPoint6[6901] = {X 226.6792, Y 41.8070, Z -8.0000, A 0.000, B 0.000, C 0.000 }
gfCNCPoint6[6902] = {X 227.1174, Y 42.5436, Z -8.0000, A 0.000, B 0.000, C 0.000 }
gfCNCPoint6[6903] = {X 227.3887, Y 43.3567, Z -8.0000, A 0.000, B 0.000, C 0.000 }
gfCNCPoint6[6904] = {X 227.4805, Y 44.2089, Z -8.0000, A 0.000, B 0.000, C 0.000 }
gfCNCPoint6[6905] = {X 227.4805, Y 45.0000, Z -8.0000, A 0.000, B 0.000, C 0.000 }
gfCNCPoint6[6906] = {X 227.3802, Y 45.8901, Z -8.0000, A 0.000, B 0.000, C 0.000 }
gfCNCPoint6[6907] = {X 227.0844, Y 46.7355, Z -8.0000, A 0.000, B 0.000, C 0.000 }
gfCNCPoint6[6908] = {X 226.6078, Y 47.4940, Z -8.0000, A 0.000, B 0.000, C 0.000 }
gfCNCPoint6[6909] = {X 225.9744, Y 48.1273, Z -8.0000, A 0.000, B 0.000, C 0.000 }
gfCNCPoint6[6910] = {X 225.2160, Y 48.6039, Z -8.0000, A 0.000, B 0.000, C 0.000 }
gfCNCPoint6[6911] = {X 224.3706, Y 48.8997, Z -8.0000, A 0.000, B 0.000, C 0.000 }
gfCNCPoint6[6912] = {X 223.4805, Y 49.0000, Z -8.0000, A 0.000, B 0.000, C 0.000 }
gfCNCPoint6[6913] = {X 217.0370, Y 49.0000, Z -8.0000, A 0.000, B 0.000, C 0.000 }
gfCNCPoint6[6914] = {X 216.1469, Y 48.8997, Z -8.0000, A 0.000, B 0.000, C 0.000 }
gfCNCPoint6[6915] = {X 215.3015, Y 48.6039, Z -8.0000, A 0.000, B 0.000, C 0.000 }
gfCNCPoint6[6916] = {X 214.5430, Y 48.1273, Z -8.0000, A 0.000, B 0.000, C 0.000 }
gfCNCPoint6[6917] = {X 213.9097, Y 47.4939, Z -8.0000, A 0.000, B 0.000, C 0.000 }
gfCNCPoint6[6918] = {X 213.4331, Y 46.7355, Z -8.0000, A 0.000, B 0.000, C 0.000 }
gfCNCPoint6[6919] = {X 213.1373, Y 45.8901, Z -8.0000, A 0.000, B 0.000, C 0.000 }
gfCNCPoint6[6920] = {X 213.0370, Y 45.0000, Z -8.0000, A 0.000, B 0.000, C 0.000 }
gfCNCPoint6[6921] = {X 213.0370, Y 44.1900, Z -8.0000, A 0.000, B 0.000, C 0.000 }
gfCNCPoint6[6922] = {X 213.1545, Y 43.2375, Z -8.0000, A 0.000, B 0.000, C 0.000 }
gfCNCPoint6[6923] = {X 213.5000, Y 42.3421, Z -8.0000, A 0.000, B 0.000, C 0.000 }
gfCNCPoint6[6924] = {X 214.0527, Y 41.5574, Z -8.0000, A 0.000, B 0.000, C 0.000 }
gfCNCPoint6[6925] = {X 214.5582, Y 40.9999, Z -8.0000, A 0.000, B 0.000, C 0.000 }
gfCNCPoint6[6926] = {X 214.5635, Y 40.3075, Z -8.0000, A 0.000, B 0.000, C 0.000 }
gfCNCPoint6[6927] = {X 214.5635, Y 28.5736, Z -8.0000, A 0.000, B 0.000, C 0.000 }
gfCNCPoint6[6928] = {X 210.4835, Y 28.5736, Z -8.0000, A 0.000, B 0.000, C 0.000 }
gfCNCPoint6[6929] = {X 210.4835, Y 28.5736, Z -5.0000, A 0.000, B 0.000, C 0.000 }
gfCNCPoint6[6930] = {X 210.4835, Y 28.5736, Z 11.0000, A 0.000, B 0.000, C 0.000 }
gfCNCPoint6[6931] = {X 273.6049, Y 28.5937, Z 11.0000, A 0.000, B 0.000, C 0.000 }
gfCNCPoint6[6932] = {X 273.6049, Y 28.5937, Z -5.0000, A 0.000, B 0.000, C 0.000 }
gfCNCPoint6[6933] = {X 273.6049, Y 28.5937, Z -8.0000, A 0.000, B 0.000, C 0.000 }
gfCNCPoint6[6934] = {X 269.5249, Y 28.5938, Z -8.0000, A 0.000, B 0.000, C 0.000 }
gfCNCPoint6[6935] = {X 269.5251, Y 40.9143, Z -8.0000, A 0.000, B 0.000, C 0.000 }
gfCNCPoint6[6936] = {X 269.5383, Y 40.9253, Z -8.0000, A 0.000, B 0.000, C 0.000 }
gfCNCPoint6[6937] = {X 270.1704, Y 41.5947, Z -8.0000, A 0.000, B 0.000, C 0.000 }
gfCNCPoint6[6938] = {X 270.6462, Y 42.3829, Z -8.0000, A 0.000, B 0.000, C 0.000 }
gfCNCPoint6[6939] = {X 270.9442, Y 43.2541, Z -8.0000, A 0.000, B 0.000, C 0.000 }
gfCNCPoint6[6940] = {X 271.0508, Y 44.1686, Z -8.0000, A 0.000, B 0.000, C 0.000 }
gfCNCPoint6[6941] = {X 271.0510, Y 45.0000, Z -8.0000, A 0.000, B 0.000, C 0.000 }
gfCNCPoint6[6942] = {X 270.9427, Y 45.9613, Z -8.0000, A 0.000, B 0.000, C 0.000 }
gfCNCPoint6[6943] = {X 270.6232, Y 46.8744, Z -8.0000, A 0.000, B 0.000, C 0.000 }
gfCNCPoint6[6944] = {X 270.1085, Y 47.6935, Z -8.0000, A 0.000, B 0.000, C 0.000 }
gfCNCPoint6[6945] = {X 269.4245, Y 48.3775, Z -8.0000, A 0.000, B 0.000, C 0.000 }
gfCNCPoint6[6946] = {X 268.6054, Y 48.8922, Z -8.0000, A 0.000, B 0.000, C 0.000 }
gfCNCPoint6[6947] = {X 267.6923, Y 49.2117, Z -8.0000, A 0.000, B 0.000, C 0.000 }
gfCNCPoint6[6948] = {X 266.7310, Y 49.3200, Z -8.0000, A 0.000, B 0.000, C 0.000 }
gfCNCPoint6[6949] = {X 260.2876, Y 49.3200, Z -8.0000, A 0.000, B 0.000, C 0.000 }
gfCNCPoint6[6950] = {X 259.3310, Y 49.2128, Z -8.0000, A 0.000, B 0.000, C 0.000 }
gfCNCPoint6[6951] = {X 258.4219, Y 48.8963, Z -8.0000, A 0.000, B 0.000, C 0.000 }
gfCNCPoint6[6952] = {X 257.6054, Y 48.3865, Z -8.0000, A 0.000, B 0.000, C 0.000 }
gfCNCPoint6[6953] = {X 256.9221, Y 47.7085, Z -8.0000, A 0.000, B 0.000, C 0.000 }
gfCNCPoint6[6954] = {X 256.4059, Y 46.8960, Z -8.0000, A 0.000, B 0.000, C 0.000 }
gfCNCPoint6[6955] = {X 256.0824, Y 45.9894, Z -8.0000, A 0.000, B 0.000, C 0.000 }
gfCNCPoint6[6956] = {X 255.9677, Y 45.0336, Z -8.0000, A 0.000, B 0.000, C 0.000 }
gfCNCPoint6[6957] = {X 255.9680, Y 44.1494, Z -8.0000, A 0.000, B 0.000, C 0.000 }
gfCNCPoint6[6958] = {X 256.0784, Y 43.2364, Z -8.0000, A 0.000, B 0.000, C 0.000 }
gfCNCPoint6[6959] = {X 256.3796, Y 42.3675, Z -8.0000, A 0.000, B 0.000, C 0.000 }
gfCNCPoint6[6960] = {X 256.8579, Y 41.5821, Z -8.0000, A 0.000, B 0.000, C 0.000 }
gfCNCPoint6[6961] = {X 257.4915, Y 40.9157, Z -8.0000, A 0.000, B 0.000, C 0.000 }
gfCNCPoint6[6962] = {X 257.4915, Y 34.4738, Z -8.0000, A 0.000, B 0.000, C 0.000 }
gfCNCPoint6[6963] = {X 254.7690, Y 34.4738, Z -8.0000, A 0.000, B 0.000, C 0.000 }
gfCNCPoint6[6964] = {X 250.4841, Y 42.8195, Z -8.0000, A 0.000, B 0.000, C 0.000 }
gfCNCPoint6[6965] = {X 250.6528, Y 43.4867, Z -8.0000, A 0.000, B 0.000, C 0.000 }
gfCNCPoint6[6966] = {X 250.7134, Y 44.1723, Z -8.0000, A 0.000, B 0.000, C 0.000 }
gfCNCPoint6[6967] = {X 250.7136, Y 45.0000, Z -8.0000, A 0.000, B 0.000, C 0.000 }
gfCNCPoint6[6968] = {X 250.6052, Y 45.9613, Z -8.0000, A 0.000, B 0.000, C 0.000 }
gfCNCPoint6[6969] = {X 250.2857, Y 46.8744, Z -8.0000, A 0.000, B 0.000, C 0.000 }
gfCNCPoint6[6970] = {X 249.7711, Y 47.6935, Z -8.0000, A 0.000, B 0.000, C 0.000 }
gfCNCPoint6[6971] = {X 249.0870, Y 48.3775, Z -8.0000, A 0.000, B 0.000, C 0.000 }
gfCNCPoint6[6972] = {X 248.2679, Y 48.8922, Z -8.0000, A 0.000, B 0.000, C 0.000 }
gfCNCPoint6[6973] = {X 247.3548, Y 49.2117, Z -8.0000, A 0.000, B 0.000, C 0.000 }
gfCNCPoint6[6974] = {X 246.3936, Y 49.3200, Z -8.0000, A 0.000, B 0.000, C 0.000 }
gfCNCPoint6[6975] = {X 239.8075, Y 49.3200, Z -8.0000, A 0.000, B 0.000, C 0.000 }
gfCNCPoint6[6976] = {X 238.8462, Y 49.2117, Z -8.0000, A 0.000, B 0.000, C 0.000 }
gfCNCPoint6[6977] = {X 237.9331, Y 48.8922, Z -8.0000, A 0.000, B 0.000, C 0.000 }
gfCNCPoint6[6978] = {X 237.1141, Y 48.3775, Z -8.0000, A 0.000, B 0.000, C 0.000 }
gfCNCPoint6[6979] = {X 236.4300, Y 47.6935, Z -8.0000, A 0.000, B 0.000, C 0.000 }
gfCNCPoint6[6980] = {X 235.9153, Y 46.8745, Z -8.0000, A 0.000, B 0.000, C 0.000 }
gfCNCPoint6[6981] = {X 235.5958, Y 45.9614, Z -8.0000, A 0.000, B 0.000, C 0.000 }
gfCNCPoint6[6982] = {X 235.4875, Y 45.0001, Z -8.0000, A 0.000, B 0.000, C 0.000 }
gfCNCPoint6[6983] = {X 235.4879, Y 44.1494, Z -8.0000, A 0.000, B 0.000, C 0.000 }
gfCNCPoint6[6984] = {X 235.5856, Y 43.2935, Z -8.0000, A 0.000, B 0.000, C 0.000 }
gfCNCPoint6[6985] = {X 235.8511, Y 42.4740, Z -8.0000, A 0.000, B 0.000, C 0.000 }
gfCNCPoint6[6986] = {X 236.2739, Y 41.7236, Z -8.0000, A 0.000, B 0.000, C 0.000 }
gfCNCPoint6[6987] = {X 236.8373, Y 41.0719, Z -8.0000, A 0.000, B 0.000, C 0.000 }
gfCNCPoint6[6988] = {X 237.5187, Y 40.5449, Z -8.0000, A 0.000, B 0.000, C 0.000 }
gfCNCPoint6[6989] = {X 238.2911, Y 40.1637, Z -8.0000, A 0.000, B 0.000, C 0.000 }
gfCNCPoint6[6990] = {X 242.2798, Y 32.3564, Z -8.0000, A 0.000, B 0.000, C 0.000 }
gfCNCPoint6[6991] = {X 241.1097, Y 31.5697, Z -8.0000, A 0.000, B 0.000, C 0.000 }
gfCNCPoint6[6992] = {X 240.0464, Y 30.6437, Z -8.0000, A 0.000, B 0.000, C 0.000 }
gfCNCPoint6[6993] = {X 239.1065, Y 29.5928, Z -8.0000, A 0.000, B 0.000, C 0.000 }
gfCNCPoint6[6994] = {X 238.3044, Y 28.4333, Z -8.0000, A 0.000, B 0.000, C 0.000 }
gfCNCPoint6[6995] = {X 237.6526, Y 27.1830, Z -8.0000, A 0.000, B 0.000, C 0.000 }
gfCNCPoint6[6996] = {X 237.1613, Y 25.8615, Z -8.0000, A 0.000, B 0.000, C 0.000 }
gfCNCPoint6[6997] = {X 236.7411, Y 24.0500, Z -8.0000, A 0.000, B 0.000, C 0.000 }
gfCNCPoint6[6998] = {X 236.5270, Y 22.2028, Z -8.0000, A 0.000, B 0.000, C 0.000 }
gfCNCPoint6[6999] = {X 236.5216, Y 20.3433, Z -8.0000, A 0.000, B 0.000, C 0.000 }
gfCNCPoint6[7000] = {X 236.7251, Y 18.4949, Z -8.0000, A 0.000, B 0.000, C 0.000 }
gfCNCPoint6[7001] = {X 237.1348, Y 16.6810, Z -8.0000, A 0.000, B 0.000, C 0.000 }
gfCNCPoint6[7002] = {X 237.7054, Y 15.1052, Z -8.0000, A 0.000, B 0.000, C 0.000 }
gfCNCPoint6[7003] = {X 238.4925, Y 13.6255, Z -8.0000, A 0.000, B 0.000, C 0.000 }
gfCNCPoint6[7004] = {X 239.4805, Y 12.2717, Z -8.0000, A 0.000, B 0.000, C 0.000 }
gfCNCPoint6[7005] = {X 240.6496, Y 11.0709, Z -8.0000, A 0.000, B 0.000, C 0.000 }
gfCNCPoint6[7006] = {X 241.9764, Y 10.0469, Z -8.0000, A 0.000, B 0.000, C 0.000 }
gfCNCPoint6[7007] = {X 243.4344, Y 9.2203, Z -8.0000, A 0.000, B 0.000, C 0.000 }
gfCNCPoint6[7008] = {X 244.9943, Y 8.6077, Z -8.0000, A 0.000, B 0.000, C 0.000 }
gfCNCPoint6[7009] = {X 246.6252, Y 8.2213, Z -8.0000, A 0.000, B 0.000, C 0.000 }
gfCNCPoint6[7010] = {X 248.7221, Y 7.9498, Z -8.0000, A 0.000, B 0.000, C 0.000 }
gfCNCPoint6[7011] = {X 250.8349, Y 7.8692, Z -8.0000, A 0.000, B 0.000, C 0.000 }
gfCNCPoint6[7012] = {X 266.7633, Y 7.8692, Z -8.0000, A 0.000, B 0.000, C 0.000 }
gfCNCPoint6[7013] = {X 267.7187, Y 7.9840, Z -8.0000, A 0.000, B 0.000, C 0.000 }
gfCNCPoint6[7014] = {X 268.6251, Y 8.3073, Z -8.0000, A 0.000, B 0.000, C 0.000 }
gfCNCPoint6[7015] = {X 269.4374, Y 8.8231, Z -8.0000, A 0.000, B 0.000, C 0.000 }
gfCNCPoint6[7016] = {X 270.1155, Y 9.5059, Z -8.0000, A 0.000, B 0.000, C 0.000 }
gfCNCPoint6[7017] = {X 270.6257, Y 10.3218, Z -8.0000, A 0.000, B 0.000, C 0.000 }
gfCNCPoint6[7018] = {X 270.9428, Y 11.2303, Z -8.0000, A 0.000, B 0.000, C 0.000 }
gfCNCPoint6[7019] = {X 271.0510, Y 12.1865, Z -8.0000, A 0.000, B 0.000, C 0.000 }
gfCNCPoint6[7020] = {X 271.0508, Y 13.0225, Z -8.0000, A 0.000, B 0.000, C 0.000 }
gfCNCPoint6[7021] = {X 270.9425, Y 13.9402, Z -8.0000, A 0.000, B 0.000, C 0.000 }
gfCNCPoint6[7022] = {X 270.6415, Y 14.8139, Z -8.0000, A 0.000, B 0.000, C 0.000 }
gfCNCPoint6[7023] = {X 270.1616, Y 15.6036, Z -8.0000, A 0.000, B 0.000, C 0.000 }
gfCNCPoint6[7024] = {X 269.5247, Y 16.2732, Z -8.0000, A 0.000, B 0.000, C 0.000 }
gfCNCPoint6[7025] = {X 269.5249, Y 28.5938, Z -8.0000, A 0.000, B 0.000, C 0.000 }
gfCNCPoint6[7026] = {X 273.5249, Y 28.5937, Z -8.0000, A 0.000, B 0.000, C 0.000 }
gfCNCPoint6[7027] = {X 269.4449, Y 28.5938, Z -8.0000, A 0.000, B 0.000, C 0.000 }
gfCNCPoint6[7028] = {X 269.4451, Y 40.9521, Z -8.0000, A 0.000, B 0.000, C 0.000 }
gfCNCPoint6[7029] = {X 269.4869, Y 40.9866, Z -8.0000, A 0.000, B 0.000, C 0.000 }
gfCNCPoint6[7030] = {X 270.1070, Y 41.6436, Z -8.0000, A 0.000, B 0.000, C 0.000 }
gfCNCPoint6[7031] = {X 270.5739, Y 42.4171, Z -8.0000, A 0.000, B 0.000, C 0.000 }
gfCNCPoint6[7032] = {X 270.8662, Y 43.2719, Z -8.0000, A 0.000, B 0.000, C 0.000 }
gfCNCPoint6[7033] = {X 270.9708, Y 44.1693, Z -8.0000, A 0.000, B 0.000, C 0.000 }
gfCNCPoint6[7034] = {X 270.9710, Y 45.0000, Z -8.0000, A 0.000, B 0.000, C 0.000 }
gfCNCPoint6[7035] = {X 270.8647, Y 45.9435, Z -8.0000, A 0.000, B 0.000, C 0.000 }
gfCNCPoint6[7036] = {X 270.5511, Y 46.8397, Z -8.0000, A 0.000, B 0.000, C 0.000 }
gfCNCPoint6[7037] = {X 270.0460, Y 47.6436, Z -8.0000, A 0.000, B 0.000, C 0.000 }
gfCNCPoint6[7038] = {X 269.3746, Y 48.3150, Z -8.0000, A 0.000, B 0.000, C 0.000 }
gfCNCPoint6[7039] = {X 268.5707, Y 48.8201, Z -8.0000, A 0.000, B 0.000, C 0.000 }
gfCNCPoint6[7040] = {X 267.6745, Y 49.1337, Z -8.0000, A 0.000, B 0.000, C 0.000 }
gfCNCPoint6[7041] = {X 266.7310, Y 49.2400, Z -8.0000, A 0.000, B 0.000, C 0.000 }
gfCNCPoint6[7042] = {X 260.2876, Y 49.2400, Z -8.0000, A 0.000, B 0.000, C 0.000 }
gfCNCPoint6[7043] = {X 259.3487, Y 49.1347, Z -8.0000, A 0.000, B 0.000, C 0.000 }
gfCNCPoint6[7044] = {X 258.4564, Y 48.8242, Z -8.0000, A 0.000, B 0.000, C 0.000 }
gfCNCPoint6[7045] = {X 257.6550, Y 48.3238, Z -8.0000, A 0.000, B 0.000, C 0.000 }
gfCNCPoint6[7046] = {X 256.9844, Y 47.6583, Z -8.0000, A 0.000, B 0.000, C 0.000 }
gfCNCPoint6[7047] = {X 256.4777, Y 46.8609, Z -8.0000, A 0.000, B 0.000, C 0.000 }
gfCNCPoint6[7048] = {X 256.1603, Y 45.9711, Z -8.0000, A 0.000, B 0.000, C 0.000 }
gfCNCPoint6[7049] = {X 256.0477, Y 45.0330, Z -8.0000, A 0.000, B 0.000, C 0.000 }
gfCNCPoint6[7050] = {X 256.0480, Y 44.1505, Z -8.0000, A 0.000, B 0.000, C 0.000 }
gfCNCPoint6[7051] = {X 256.1585, Y 43.2454, Z -8.0000, A 0.000, B 0.000, C 0.000 }
gfCNCPoint6[7052] = {X 256.4599, Y 42.3850, Z -8.0000, A 0.000, B 0.000, C 0.000 }
gfCNCPoint6[7053] = {X 256.9383, Y 41.6088, Z -8.0000, A 0.000, B 0.000, C 0.000 }
gfCNCPoint6[7054] = {X 257.5715, Y 40.9529, Z -8.0000, A 0.000, B 0.000, C 0.000 }
gfCNCPoint6[7055] = {X 257.5715, Y 34.3938, Z -8.0000, A 0.000, B 0.000, C 0.000 }
gfCNCPoint6[7056] = {X 254.7201, Y 34.3938, Z -8.0000, A 0.000, B 0.000, C 0.000 }
gfCNCPoint6[7057] = {X 250.3973, Y 42.8133, Z -8.0000, A 0.000, B 0.000, C 0.000 }
gfCNCPoint6[7058] = {X 250.5711, Y 43.4834, Z -8.0000, A 0.000, B 0.000, C 0.000 }
gfCNCPoint6[7059] = {X 250.6334, Y 44.1730, Z -8.0000, A 0.000, B 0.000, C 0.000 }
gfCNCPoint6[7060] = {X 250.6336, Y 45.0000, Z -8.0000, A 0.000, B 0.000, C 0.000 }
gfCNCPoint6[7061] = {X 250.5273, Y 45.9435, Z -8.0000, A 0.000, B 0.000, C 0.000 }
gfCNCPoint6[7062] = {X 250.2137, Y 46.8397, Z -8.0000, A 0.000, B 0.000, C 0.000 }
gfCNCPoint6[7063] = {X 249.7085, Y 47.6436, Z -8.0000, A 0.000, B 0.000, C 0.000 }
gfCNCPoint6[7064] = {X 249.0372, Y 48.3150, Z -8.0000, A 0.000, B 0.000, C 0.000 }
gfCNCPoint6[7065] = {X 248.2332, Y 48.8201, Z -8.0000, A 0.000, B 0.000, C 0.000 }
gfCNCPoint6[7066] = {X 247.3370, Y 49.1337, Z -8.0000, A 0.000, B 0.000, C 0.000 }
gfCNCPoint6[7067] = {X 246.3936, Y 49.2400, Z -8.0000, A 0.000, B 0.000, C 0.000 }
gfCNCPoint6[7068] = {X 239.8075, Y 49.2400, Z -8.0000, A 0.000, B 0.000, C 0.000 }
gfCNCPoint6[7069] = {X 238.8640, Y 49.1337, Z -8.0000, A 0.000, B 0.000, C 0.000 }
gfCNCPoint6[7070] = {X 237.9679, Y 48.8201, Z -8.0000, A 0.000, B 0.000, C 0.000 }
gfCNCPoint6[7071] = {X 237.1639, Y 48.3150, Z -8.0000, A 0.000, B 0.000, C 0.000 }
gfCNCPoint6[7072] = {X 236.4926, Y 47.6436, Z -8.0000, A 0.000, B 0.000, C 0.000 }
gfCNCPoint6[7073] = {X 235.9874, Y 46.8397, Z -8.0000, A 0.000, B 0.000, C 0.000 }
gfCNCPoint6[7074] = {X 235.6738, Y 45.9436, Z -8.0000, A 0.000, B 0.000, C 0.000 }
gfCNCPoint6[7075] = {X 235.5675, Y 45.0001, Z -8.0000, A 0.000, B 0.000, C 0.000 }
gfCNCPoint6[7076] = {X 235.5679, Y 44.1505, Z -8.0000, A 0.000, B 0.000, C 0.000 }
gfCNCPoint6[7077] = {X 235.6649, Y 43.3054, Z -8.0000, A 0.000, B 0.000, C 0.000 }
gfCNCPoint6[7078] = {X 235.9285, Y 42.4967, Z -8.0000, A 0.000, B 0.000, C 0.000 }
gfCNCPoint6[7079] = {X 236.3483, Y 41.7570, Z -8.0000, A 0.000, B 0.000, C 0.000 }
gfCNCPoint6[7080] = {X 236.9073, Y 41.1158, Z -8.0000, A 0.000, B 0.000, C 0.000 }
gfCNCPoint6[7081] = {X 237.5830, Y 40.5992, Z -8.0000, A 0.000, B 0.000, C 0.000 }
gfCNCPoint6[7082] = {X 238.3482, Y 40.2278, Z -8.0000, A 0.000, B 0.000, C 0.000 }
gfCNCPoint6[7083] = {X 242.3855, Y 32.3253, Z -8.0000, A 0.000, B 0.000, C 0.000 }
gfCNCPoint6[7084] = {X 241.2084, Y 31.5444, Z -8.0000, A 0.000, B 0.000, C 0.000 }
gfCNCPoint6[7085] = {X 240.1386, Y 30.6221, Z -8.0000, A 0.000, B 0.000, C 0.000 }
gfCNCPoint6[7086] = {X 239.1928, Y 29.5729, Z -8.0000, A 0.000, B 0.000, C 0.000 }
gfCNCPoint6[7087] = {X 238.3859, Y 28.4135, Z -8.0000, A 0.000, B 0.000, C 0.000 }
gfCNCPoint6[7088] = {X 237.7309, Y 27.1621, Z -8.0000, A 0.000, B 0.000, C 0.000 }
gfCNCPoint6[7089] = {X 237.2379, Y 25.8383, Z -8.0000, A 0.000, B 0.000, C 0.000 }
gfCNCPoint6[7090] = {X 236.8198, Y 24.0358, Z -8.0000, A 0.000, B 0.000, C 0.000 }
gfCNCPoint6[7091] = {X 236.6068, Y 22.1976, Z -8.0000, A 0.000, B 0.000, C 0.000 }
gfCNCPoint6[7092] = {X 236.6015, Y 20.3472, Z -8.0000, A 0.000, B 0.000, C 0.000 }
gfCNCPoint6[7093] = {X 236.8040, Y 18.5079, Z -8.0000, A 0.000, B 0.000, C 0.000 }
gfCNCPoint6[7094] = {X 237.2117, Y 16.7030, Z -8.0000, A 0.000, B 0.000, C 0.000 }
gfCNCPoint6[7095] = {X 237.7785, Y 15.1377, Z -8.0000, A 0.000, B 0.000, C 0.000 }
gfCNCPoint6[7096] = {X 238.5603, Y 13.6680, Z -8.0000, A 0.000, B 0.000, C 0.000 }
gfCNCPoint6[7097] = {X 239.5417, Y 12.3233, Z -8.0000, A 0.000, B 0.000, C 0.000 }
gfCNCPoint6[7098] = {X 240.7030, Y 11.1305, Z -8.0000, A 0.000, B 0.000, C 0.000 }
gfCNCPoint6[7099] = {X 242.0209, Y 10.1134, Z -8.0000, A 0.000, B 0.000, C 0.000 }
gfCNCPoint6[7100] = {X 243.4691, Y 9.2924, Z -8.0000, A 0.000, B 0.000, C 0.000 }
gfCNCPoint6[7101] = {X 245.0187, Y 8.6839, Z -8.0000, A 0.000, B 0.000, C 0.000 }
gfCNCPoint6[7102] = {X 246.6385, Y 8.3001, Z -8.0000, A 0.000, B 0.000, C 0.000 }
gfCNCPoint6[7103] = {X 248.7286, Y 8.0295, Z -8.0000, A 0.000, B 0.000, C 0.000 }
gfCNCPoint6[7104] = {X 250.8346, Y 7.9492, Z -8.0000, A 0.000, B 0.000, C 0.000 }
gfCNCPoint6[7105] = {X 266.7627, Y 7.9492, Z -8.0000, A 0.000, B 0.000, C 0.000 }
gfCNCPoint6[7106] = {X 267.7004, Y 8.0619, Z -8.0000, A 0.000, B 0.000, C 0.000 }
gfCNCPoint6[7107] = {X 268.5900, Y 8.3792, Z -8.0000, A 0.000, B 0.000, C 0.000 }
gfCNCPoint6[7108] = {X 269.3873, Y 8.8855, Z -8.0000, A 0.000, B 0.000, C 0.000 }
gfCNCPoint6[7109] = {X 270.0528, Y 9.5556, Z -8.0000, A 0.000, B 0.000, C 0.000 }
gfCNCPoint6[7110] = {X 270.5536, Y 10.3564, Z -8.0000, A 0.000, B 0.000, C 0.000 }
gfCNCPoint6[7111] = {X 270.8648, Y 11.2481, Z -8.0000, A 0.000, B 0.000, C 0.000 }
gfCNCPoint6[7112] = {X 270.9710, Y 12.1866, Z -8.0000, A 0.000, B 0.000, C 0.000 }
gfCNCPoint6[7113] = {X 270.9708, Y 13.0217, Z -8.0000, A 0.000, B 0.000, C 0.000 }
gfCNCPoint6[7114] = {X 270.8625, Y 13.9314, Z -8.0000, A 0.000, B 0.000, C 0.000 }
gfCNCPoint6[7115] = {X 270.5612, Y 14.7966, Z -8.0000, A 0.000, B 0.000, C 0.000 }
gfCNCPoint6[7116] = {X 270.0811, Y 15.5769, Z -8.0000, A 0.000, B 0.000, C 0.000 }
gfCNCPoint6[7117] = {X 269.4447, Y 16.2359, Z -8.0000, A 0.000, B 0.000, C 0.000 }
gfCNCPoint6[7118] = {X 269.4449, Y 28.5938, Z -8.0000, A 0.000, B 0.000, C 0.000 }
gfCNCPoint6[7119] = {X 273.4449, Y 28.5937, Z -8.0000, A 0.000, B 0.000, C 0.000 }
gfCNCPoint6[7120] = {X 269.3649, Y 28.5938, Z -8.0000, A 0.000, B 0.000, C 0.000 }
gfCNCPoint6[7121] = {X 269.3651, Y 40.9898, Z -8.0000, A 0.000, B 0.000, C 0.000 }
gfCNCPoint6[7122] = {X 269.4354, Y 41.0478, Z -8.0000, A 0.000, B 0.000, C 0.000 }
gfCNCPoint6[7123] = {X 270.0436, Y 41.6924, Z -8.0000, A 0.000, B 0.000, C 0.000 }
gfCNCPoint6[7124] = {X 270.5015, Y 42.4512, Z -8.0000, A 0.000, B 0.000, C 0.000 }
gfCNCPoint6[7125] = {X 270.7882, Y 43.2898, Z -8.0000, A 0.000, B 0.000, C 0.000 }
gfCNCPoint6[7126] = {X 270.8909, Y 44.1700, Z -8.0000, A 0.000, B 0.000, C 0.000 }
gfCNCPoint6[7127] = {X 270.8910, Y 45.0000, Z -8.0000, A 0.000, B 0.000, C 0.000 }
gfCNCPoint6[7128] = {X 270.7867, Y 45.9257, Z -8.0000, A 0.000, B 0.000, C 0.000 }
gfCNCPoint6[7129] = {X 270.4791, Y 46.8050, Z -8.0000, A 0.000, B 0.000, C 0.000 }
gfCNCPoint6[7130] = {X 269.9835, Y 47.5937, Z -8.0000, A 0.000, B 0.000, C 0.000 }
gfCNCPoint6[7131] = {X 269.3247, Y 48.2524, Z -8.0000, A 0.000, B 0.000, C 0.000 }
gfCNCPoint6[7132] = {X 268.5360, Y 48.7480, Z -8.0000, A 0.000, B 0.000, C 0.000 }
gfCNCPoint6[7133] = {X 267.6567, Y 49.0557, Z -8.0000, A 0.000, B 0.000, C 0.000 }
gfCNCPoint6[7134] = {X 266.7310, Y 49.1600, Z -8.0000, A 0.000, B 0.000, C 0.000 }
gfCNCPoint6[7135] = {X 260.2876, Y 49.1600, Z -8.0000, A 0.000, B 0.000, C 0.000 }
gfCNCPoint6[7136] = {X 259.3664, Y 49.0567, Z -8.0000, A 0.000, B 0.000, C 0.000 }
gfCNCPoint6[7137] = {X 258.4910, Y 48.7520, Z -8.0000, A 0.000, B 0.000, C 0.000 }
gfCNCPoint6[7138] = {X 257.7047, Y 48.2611, Z -8.0000, A 0.000, B 0.000, C 0.000 }
gfCNCPoint6[7139] = {X 257.0467, Y 47.6082, Z -8.0000, A 0.000, B 0.000, C 0.000 }
gfCNCPoint6[7140] = {X 256.5496, Y 46.8258, Z -8.0000, A 0.000, B 0.000, C 0.000 }
gfCNCPoint6[7141] = {X 256.2381, Y 45.9527, Z -8.0000, A 0.000, B 0.000, C 0.000 }
gfCNCPoint6[7142] = {X 256.1277, Y 45.0324, Z -8.0000, A 0.000, B 0.000, C 0.000 }
gfCNCPoint6[7143] = {X 256.1280, Y 44.1516, Z -8.0000, A 0.000, B 0.000, C 0.000 }
gfCNCPoint6[7144] = {X 256.2385, Y 43.2545, Z -8.0000, A 0.000, B 0.000, C 0.000 }
gfCNCPoint6[7145] = {X 256.5401, Y 42.4026, Z -8.0000, A 0.000, B 0.000, C 0.000 }
gfCNCPoint6[7146] = {X 257.0187, Y 41.6358, Z -8.0000, A 0.000, B 0.000, C 0.000 }
gfCNCPoint6[7147] = {X 257.6515, Y 40.9906, Z -8.0000, A 0.000, B 0.000, C 0.000 }
gfCNCPoint6[7148] = {X 257.6515, Y 34.3138, Z -8.0000, A 0.000, B 0.000, C 0.000 }
gfCNCPoint6[7149] = {X 254.6713, Y 34.3138, Z -8.0000, A 0.000, B 0.000, C 0.000 }
gfCNCPoint6[7150] = {X 250.3104, Y 42.8074, Z -8.0000, A 0.000, B 0.000, C 0.000 }
gfCNCPoint6[7151] = {X 250.4893, Y 43.4803, Z -8.0000, A 0.000, B 0.000, C 0.000 }
gfCNCPoint6[7152] = {X 250.5534, Y 44.1736, Z -8.0000, A 0.000, B 0.000, C 0.000 }
gfCNCPoint6[7153] = {X 250.5536, Y 45.0000, Z -8.0000, A 0.000, B 0.000, C 0.000 }
gfCNCPoint6[7154] = {X 250.4493, Y 45.9257, Z -8.0000, A 0.000, B 0.000, C 0.000 }
gfCNCPoint6[7155] = {X 250.1416, Y 46.8050, Z -8.0000, A 0.000, B 0.000, C 0.000 }
gfCNCPoint6[7156] = {X 249.6460, Y 47.5937, Z -8.0000, A 0.000, B 0.000, C 0.000 }
gfCNCPoint6[7157] = {X 248.9873, Y 48.2524, Z -8.0000, A 0.000, B 0.000, C 0.000 }
gfCNCPoint6[7158] = {X 248.1985, Y 48.7480, Z -8.0000, A 0.000, B 0.000, C 0.000 }
gfCNCPoint6[7159] = {X 247.3192, Y 49.0557, Z -8.0000, A 0.000, B 0.000, C 0.000 }
gfCNCPoint6[7160] = {X 246.3936, Y 49.1600, Z -8.0000, A 0.000, B 0.000, C 0.000 }
gfCNCPoint6[7161] = {X 239.8075, Y 49.1600, Z -8.0000, A 0.000, B 0.000, C 0.000 }
gfCNCPoint6[7162] = {X 238.8818, Y 49.0557, Z -8.0000, A 0.000, B 0.000, C 0.000 }
gfCNCPoint6[7163] = {X 238.0026, Y 48.7480, Z -8.0000, A 0.000, B 0.000, C 0.000 }
gfCNCPoint6[7164] = {X 237.2138, Y 48.2524, Z -8.0000, A 0.000, B 0.000, C 0.000 }
gfCNCPoint6[7165] = {X 236.5551, Y 47.5937, Z -8.0000, A 0.000, B 0.000, C 0.000 }
gfCNCPoint6[7166] = {X 236.0595, Y 46.8050, Z -8.0000, A 0.000, B 0.000, C 0.000 }
gfCNCPoint6[7167] = {X 235.7518, Y 45.9257, Z -8.0000, A 0.000, B 0.000, C 0.000 }
gfCNCPoint6[7168] = {X 235.6475, Y 45.0000, Z -8.0000, A 0.000, B 0.000, C 0.000 }
gfCNCPoint6[7169] = {X 235.6479, Y 44.1516, Z -8.0000, A 0.000, B 0.000, C 0.000 }
gfCNCPoint6[7170] = {X 235.7441, Y 43.3174, Z -8.0000, A 0.000, B 0.000, C 0.000 }
gfCNCPoint6[7171] = {X 236.0059, Y 42.5195, Z -8.0000, A 0.000, B 0.000, C 0.000 }
gfCNCPoint6[7172] = {X 236.4226, Y 41.7905, Z -8.0000, A 0.000, B 0.000, C 0.000 }
gfCNCPoint6[7173] = {X 236.9772, Y 41.1600, Z -8.0000, A 0.000, B 0.000, C 0.000 }
gfCNCPoint6[7174] = {X 237.6471, Y 40.6537, Z -8.0000, A 0.000, B 0.000, C 0.000 }
gfCNCPoint6[7175] = {X 238.4051, Y 40.2923, Z -8.0000, A 0.000, B 0.000, C 0.000 }
gfCNCPoint6[7176] = {X 242.4914, Y 32.2937, Z -8.0000, A 0.000, B 0.000, C 0.000 }
gfCNCPoint6[7177] = {X 241.3074, Y 31.5188, Z -8.0000, A 0.000, B 0.000, C 0.000 }
gfCNCPoint6[7178] = {X 240.2308, Y 30.6003, Z -8.0000, A 0.000, B 0.000, C 0.000 }
gfCNCPoint6[7179] = {X 239.2791, Y 29.5530, Z -8.0000, A 0.000, B 0.000, C 0.000 }
gfCNCPoint6[7180] = {X 238.4675, Y 28.3937, Z -8.0000, A 0.000, B 0.000, C 0.000 }
gfCNCPoint6[7181] = {X 237.8091, Y 27.1410, Z -8.0000, A 0.000, B 0.000, C 0.000 }
gfCNCPoint6[7182] = {X 237.3144, Y 25.8152, Z -8.0000, A 0.000, B 0.000, C 0.000 }
gfCNCPoint6[7183] = {X 236.8985, Y 24.0215, Z -8.0000, A 0.000, B 0.000, C 0.000 }
gfCNCPoint6[7184] = {X 236.6866, Y 22.1924, Z -8.0000, A 0.000, B 0.000, C 0.000 }
gfCNCPoint6[7185] = {X 236.6814, Y 20.3512, Z -8.0000, A 0.000, B 0.000, C 0.000 }
gfCNCPoint6[7186] = {X 236.8829, Y 18.5210, Z -8.0000, A 0.000, B 0.000, C 0.000 }
gfCNCPoint6[7187] = {X 237.2887, Y 16.7249, Z -8.0000, A 0.000, B 0.000, C 0.000 }
gfCNCPoint6[7188] = {X 237.8516, Y 15.1702, Z -8.0000, A 0.000, B 0.000, C 0.000 }
gfCNCPoint6[7189] = {X 238.6281, Y 13.7104, Z -8.0000, A 0.000, B 0.000, C 0.000 }
gfCNCPoint6[7190] = {X 239.6029, Y 12.3748, Z -8.0000, A 0.000, B 0.000, C 0.000 }
gfCNCPoint6[7191] = {X 240.7563, Y 11.1900, Z -8.0000, A 0.000, B 0.000, C 0.000 }
gfCNCPoint6[7192] = {X 242.0654, Y 10.1799, Z -8.0000, A 0.000, B 0.000, C 0.000 }
gfCNCPoint6[7193] = {X 243.5039, Y 9.3645, Z -8.0000, A 0.000, B 0.000, C 0.000 }
gfCNCPoint6[7194] = {X 245.0430, Y 8.7601, Z -8.0000, A 0.000, B 0.000, C 0.000 }
gfCNCPoint6[7195] = {X 246.6519, Y 8.3790, Z -8.0000, A 0.000, B 0.000, C 0.000 }
gfCNCPoint6[7196] = {X 248.7352, Y 8.1092, Z -8.0000, A 0.000, B 0.000, C 0.000 }
gfCNCPoint6[7197] = {X 250.8343, Y 8.0292, Z -8.0000, A 0.000, B 0.000, C 0.000 }
gfCNCPoint6[7198] = {X 266.7621, Y 8.0292, Z -8.0000, A 0.000, B 0.000, C 0.000 }
gfCNCPoint6[7199] = {X 267.6821, Y 8.1398, Z -8.0000, A 0.000, B 0.000, C 0.000 }
gfCNCPoint6[7200] = {X 268.5549, Y 8.4511, Z -8.0000, A 0.000, B 0.000, C 0.000 }
gfCNCPoint6[7201] = {X 269.3372, Y 8.9478, Z -8.0000, A 0.000, B 0.000, C 0.000 }
gfCNCPoint6[7202] = {X 269.9901, Y 9.6053, Z -8.0000, A 0.000, B 0.000, C 0.000 }
gfCNCPoint6[7203] = {X 270.4815, Y 10.3910, Z -8.0000, A 0.000, B 0.000, C 0.000 }
gfCNCPoint6[7204] = {X 270.7868, Y 11.2659, Z -8.0000, A 0.000, B 0.000, C 0.000 }
gfCNCPoint6[7205] = {X 270.8910, Y 12.1867, Z -8.0000, A 0.000, B 0.000, C 0.000 }
gfCNCPoint6[7206] = {X 270.8908, Y 13.0208, Z -8.0000, A 0.000, B 0.000, C 0.000 }
gfCNCPoint6[7207] = {X 270.7824, Y 13.9225, Z -8.0000, A 0.000, B 0.000, C 0.000 }
gfCNCPoint6[7208] = {X 270.4809, Y 14.7792, Z -8.0000, A 0.000, B 0.000, C 0.000 }
gfCNCPoint6[7209] = {X 270.0007, Y 15.5500, Z -8.0000, A 0.000, B 0.000, C 0.000 }
gfCNCPoint6[7210] = {X 269.3647, Y 16.1982, Z -8.0000, A 0.000, B 0.000, C 0.000 }
gfCNCPoint6[7211] = {X 269.3649, Y 28.5938, Z -8.0000, A 0.000, B 0.000, C 0.000 }
gfCNCPoint6[7212] = {X 273.3649, Y 28.5937, Z -8.0000, A 0.000, B 0.000, C 0.000 }
gfCNCPoint6[7213] = {X 269.2849, Y 28.5938, Z -8.0000, A 0.000, B 0.000, C 0.000 }
gfCNCPoint6[7214] = {X 269.2851, Y 41.0275, Z -8.0000, A 0.000, B 0.000, C 0.000 }
gfCNCPoint6[7215] = {X 269.3840, Y 41.1091, Z -8.0000, A 0.000, B 0.000, C 0.000 }
gfCNCPoint6[7216] = {X 269.9803, Y 41.7412, Z -8.0000, A 0.000, B 0.000, C 0.000 }
gfCNCPoint6[7217] = {X 270.4291, Y 42.4853, Z -8.0000, A 0.000, B 0.000, C 0.000 }
gfCNCPoint6[7218] = {X 270.7103, Y 43.3076, Z -8.0000, A 0.000, B 0.000, C 0.000 }
gfCNCPoint6[7219] = {X 270.8109, Y 44.1708, Z -8.0000, A 0.000, B 0.000, C 0.000 }
gfCNCPoint6[7220] = {X 270.8110, Y 45.0000, Z -8.0000, A 0.000, B 0.000, C 0.000 }
gfCNCPoint6[7221] = {X 270.7087, Y 45.9079, Z -8.0000, A 0.000, B 0.000, C 0.000 }
gfCNCPoint6[7222] = {X 270.4070, Y 46.7702, Z -8.0000, A 0.000, B 0.000, C 0.000 }
gfCNCPoint6[7223] = {X 269.9209, Y 47.5438, Z -8.0000, A 0.000, B 0.000, C 0.000 }
gfCNCPoint6[7224] = {X 269.2749, Y 48.1899, Z -8.0000, A 0.000, B 0.000, C 0.000 }
gfCNCPoint6[7225] = {X 268.5013, Y 48.6760, Z -8.0000, A 0.000, B 0.000, C 0.000 }
gfCNCPoint6[7226] = {X 267.6389, Y 48.9777, Z -8.0000, A 0.000, B 0.000, C 0.000 }
gfCNCPoint6[7227] = {X 266.7310, Y 49.0800, Z -8.0000, A 0.000, B 0.000, C 0.000 }
gfCNCPoint6[7228] = {X 260.2876, Y 49.0800, Z -8.0000, A 0.000, B 0.000, C 0.000 }
gfCNCPoint6[7229] = {X 259.3841, Y 48.9787, Z -8.0000, A 0.000, B 0.000, C 0.000 }
gfCNCPoint6[7230] = {X 258.5255, Y 48.6799, Z -8.0000, A 0.000, B 0.000, C 0.000 }
gfCNCPoint6[7231] = {X 257.7544, Y 48.1983, Z -8.0000, A 0.000, B 0.000, C 0.000 }
gfCNCPoint6[7232] = {X 257.1090, Y 47.5580, Z -8.0000, A 0.000, B 0.000, C 0.000 }
gfCNCPoint6[7233] = {X 256.6215, Y 46.7907, Z -8.0000, A 0.000, B 0.000, C 0.000 }
gfCNCPoint6[7234] = {X 256.3160, Y 45.9344, Z -8.0000, A 0.000, B 0.000, C 0.000 }
gfCNCPoint6[7235] = {X 256.2077, Y 45.0318, Z -8.0000, A 0.000, B 0.000, C 0.000 }
gfCNCPoint6[7236] = {X 256.2080, Y 44.1527, Z -8.0000, A 0.000, B 0.000, C 0.000 }
gfCNCPoint6[7237] = {X 256.3185, Y 43.2637, Z -8.0000, A 0.000, B 0.000, C 0.000 }
gfCNCPoint6[7238] = {X 256.6204, Y 42.4203, Z -8.0000, A 0.000, B 0.000, C 0.000 }
gfCNCPoint6[7239] = {X 257.0991, Y 41.6631, Z -8.0000, A 0.000, B 0.000, C 0.000 }
gfCNCPoint6[7240] = {X 257.7315, Y 41.0287, Z -8.0000, A 0.000, B 0.000, C 0.000 }
gfCNCPoint6[7241] = {X 257.7315, Y 34.2338, Z -8.0000, A 0.000, B 0.000, C 0.000 }
gfCNCPoint6[7242] = {X 254.6224, Y 34.2338, Z -8.0000, A 0.000, B 0.000, C 0.000 }
gfCNCPoint6[7243] = {X 250.2233, Y 42.8019, Z -8.0000, A 0.000, B 0.000, C 0.000 }
gfCNCPoint6[7244] = {X 250.4075, Y 43.4773, Z -8.0000, A 0.000, B 0.000, C 0.000 }
gfCNCPoint6[7245] = {X 250.4734, Y 44.1743, Z -8.0000, A 0.000, B 0.000, C 0.000 }
gfCNCPoint6[7246] = {X 250.4736, Y 45.0000, Z -8.0000, A 0.000, B 0.000, C 0.000 }
gfCNCPoint6[7247] = {X 250.3713, Y 45.9079, Z -8.0000, A 0.000, B 0.000, C 0.000 }
gfCNCPoint6[7248] = {X 250.0695, Y 46.7702, Z -8.0000, A 0.000, B 0.000, C 0.000 }
gfCNCPoint6[7249] = {X 249.5834, Y 47.5438, Z -8.0000, A 0.000, B 0.000, C 0.000 }
gfCNCPoint6[7250] = {X 248.9374, Y 48.1899, Z -8.0000, A 0.000, B 0.000, C 0.000 }
gfCNCPoint6[7251] = {X 248.1638, Y 48.6760, Z -8.0000, A 0.000, B 0.000, C 0.000 }
gfCNCPoint6[7252] = {X 247.3014, Y 48.9777, Z -8.0000, A 0.000, B 0.000, C 0.000 }
gfCNCPoint6[7253] = {X 246.3936, Y 49.0800, Z -8.0000, A 0.000, B 0.000, C 0.000 }
gfCNCPoint6[7254] = {X 239.8075, Y 49.0800, Z -8.0000, A 0.000, B 0.000, C 0.000 }
gfCNCPoint6[7255] = {X 238.8996, Y 48.9777, Z -8.0000, A 0.000, B 0.000, C 0.000 }
gfCNCPoint6[7256] = {X 238.0373, Y 48.6760, Z -8.0000, A 0.000, B 0.000, C 0.000 }
gfCNCPoint6[7257] = {X 237.2637, Y 48.1899, Z -8.0000, A 0.000, B 0.000, C 0.000 }
gfCNCPoint6[7258] = {X 236.6176, Y 47.5438, Z -8.0000, A 0.000, B 0.000, C 0.000 }
gfCNCPoint6[7259] = {X 236.1315, Y 46.7702, Z -8.0000, A 0.000, B 0.000, C 0.000 }
gfCNCPoint6[7260] = {X 235.8298, Y 45.9079, Z -8.0000, A 0.000, B 0.000, C 0.000 }
gfCNCPoint6[7261] = {X 235.7275, Y 45.0000, Z -8.0000, A 0.000, B 0.000, C 0.000 }
gfCNCPoint6[7262] = {X 235.7279, Y 44.1527, Z -8.0000, A 0.000, B 0.000, C 0.000 }
gfCNCPoint6[7263] = {X 235.8234, Y 43.3294, Z -8.0000, A 0.000, B 0.000, C 0.000 }
gfCNCPoint6[7264] = {X 236.0833, Y 42.5424, Z -8.0000, A 0.000, B 0.000, C 0.000 }
gfCNCPoint6[7265] = {X 236.4969, Y 41.8242, Z -8.0000, A 0.000, B 0.000, C 0.000 }
gfCNCPoint6[7266] = {X 237.0471, Y 41.2044, Z -8.0000, A 0.000, B 0.000, C 0.000 }
gfCNCPoint6[7267] = {X 237.7112, Y 40.7085, Z -8.0000, A 0.000, B 0.000, C 0.000 }
gfCNCPoint6[7268] = {X 238.4618, Y 40.3571, Z -8.0000, A 0.000, B 0.000, C 0.000 }
gfCNCPoint6[7269] = {X 242.5976, Y 32.2617, Z -8.0000, A 0.000, B 0.000, C 0.000 }
gfCNCPoint6[7270] = {X 241.4065, Y 31.4928, Z -8.0000, A 0.000, B 0.000, C 0.000 }
